  PROC DrawPart80()
    MoveL Offs(pOrigin,344.14,26.67,6.00),v60,z5,tPen\WObj:=wPaper;
    MoveL Offs(pOrigin,346.05,26.67,6.00),vTravel,z5,tPen\WObj:=wPaper;
    MoveL Offs(pOrigin,346.05,26.67,0.00),v60,z0,tPen\WObj:=wPaper;
    MoveL Offs(pOrigin,347.54,27.95,0.00),v40,z0,tPen\WObj:=wPaper;
    MoveL Offs(pOrigin,346.05,26.67,0.00),v40,fine,tPen\WObj:=wPaper;
    MoveL Offs(pOrigin,346.05,26.67,6.00),v60,z5,tPen\WObj:=wPaper;
    MoveL Offs(pOrigin,346.05,28.16,6.00),vTravel,z5,tPen\WObj:=wPaper;
    MoveL Offs(pOrigin,346.05,28.16,0.00),v60,z0,tPen\WObj:=wPaper;
    MoveL Offs(pOrigin,346.48,28.59,0.00),v40,z0,tPen\WObj:=wPaper;
    MoveL Offs(pOrigin,346.05,28.16,0.00),v40,fine,tPen\WObj:=wPaper;
    MoveL Offs(pOrigin,346.05,28.16,6.00),v60,z5,tPen\WObj:=wPaper;
    MoveL Offs(pOrigin,340.52,32.98,6.00),vTravel,z5,tPen\WObj:=wPaper;
    MoveL Offs(pOrigin,340.52,32.98,0.00),v60,z0,tPen\WObj:=wPaper;
    MoveL Offs(pOrigin,338.61,32.91,0.00),v40,z0,tPen\WObj:=wPaper;
    MoveL Offs(pOrigin,337.76,34.33,0.00),v40,z0,tPen\WObj:=wPaper;
    MoveL Offs(pOrigin,337.90,36.45,0.00),v40,z0,tPen\WObj:=wPaper;
    MoveL Offs(pOrigin,339.46,38.22,0.00),v40,z0,tPen\WObj:=wPaper;
    MoveL Offs(pOrigin,341.16,38.58,0.00),v40,z0,tPen\WObj:=wPaper;
    MoveL Offs(pOrigin,342.01,38.15,0.00),v40,z0,tPen\WObj:=wPaper;
    MoveL Offs(pOrigin,342.44,37.30,0.00),v40,z0,tPen\WObj:=wPaper;
    MoveL Offs(pOrigin,342.44,35.60,0.00),v40,z0,tPen\WObj:=wPaper;
    MoveL Offs(pOrigin,342.08,34.54,0.00),v40,z0,tPen\WObj:=wPaper;
    MoveL Offs(pOrigin,340.52,32.98,0.00),v40,fine,tPen\WObj:=wPaper;
    MoveL Offs(pOrigin,340.52,32.98,6.00),v60,z5,tPen\WObj:=wPaper;
    MoveL Offs(pOrigin,340.10,35.39,6.00),vTravel,z5,tPen\WObj:=wPaper;
    MoveL Offs(pOrigin,340.10,35.39,0.00),v60,z0,tPen\WObj:=wPaper;
    MoveL Offs(pOrigin,340.74,36.03,0.00),v40,fine,tPen\WObj:=wPaper;
    MoveL Offs(pOrigin,340.74,36.03,6.00),v60,z5,tPen\WObj:=wPaper;
    MoveL Offs(pOrigin,334.79,36.45,6.00),vTravel,z5,tPen\WObj:=wPaper;
    MoveL Offs(pOrigin,334.79,36.45,0.00),v60,z0,tPen\WObj:=wPaper;
    MoveL Offs(pOrigin,334.36,34.11,0.00),v40,z0,tPen\WObj:=wPaper;
    MoveL Offs(pOrigin,334.36,32.62,0.00),v40,z0,tPen\WObj:=wPaper;
    MoveL Offs(pOrigin,334.79,31.14,0.00),v40,fine,tPen\WObj:=wPaper;
    MoveL Offs(pOrigin,334.79,31.14,6.00),v60,z5,tPen\WObj:=wPaper;
    MoveL Offs(pOrigin,336.49,27.10,6.00),vTravel,z5,tPen\WObj:=wPaper;
    MoveL Offs(pOrigin,336.49,27.10,0.00),v60,z0,tPen\WObj:=wPaper;
    MoveL Offs(pOrigin,336.91,26.67,0.00),v40,z0,tPen\WObj:=wPaper;
    MoveL Offs(pOrigin,339.46,25.83,0.00),v40,z0,tPen\WObj:=wPaper;
    MoveL Offs(pOrigin,341.38,25.61,0.00),v40,z0,tPen\WObj:=wPaper;
    MoveL Offs(pOrigin,343.92,26.39,0.00),v40,z0,tPen\WObj:=wPaper;
    MoveL Offs(pOrigin,345.41,27.31,0.00),v40,z0,tPen\WObj:=wPaper;
    MoveL Offs(pOrigin,346.90,28.80,0.00),v40,z0,tPen\WObj:=wPaper;
    MoveL Offs(pOrigin,348.88,32.41,0.00),v40,z0,tPen\WObj:=wPaper;
    MoveL Offs(pOrigin,349.66,35.60,0.00),v40,z0,tPen\WObj:=wPaper;
    MoveL Offs(pOrigin,349.66,37.72,0.00),v40,z0,tPen\WObj:=wPaper;
    MoveL Offs(pOrigin,349.24,38.36,0.00),v40,z0,tPen\WObj:=wPaper;
    MoveL Offs(pOrigin,349.24,38.36,0.00),v40,z0,tPen\WObj:=wPaper;
    MoveL Offs(pOrigin,348.88,38.15,0.00),v40,z0,tPen\WObj:=wPaper;
    MoveL Offs(pOrigin,347.82,34.54,0.00),v40,z0,tPen\WObj:=wPaper;
    MoveL Offs(pOrigin,346.33,31.35,0.00),v40,z0,tPen\WObj:=wPaper;
    MoveL Offs(pOrigin,343.92,28.38,0.00),v40,z0,tPen\WObj:=wPaper;
    MoveL Offs(pOrigin,340.95,27.10,0.00),v40,z0,tPen\WObj:=wPaper;
    MoveL Offs(pOrigin,337.12,27.52,0.00),v40,z0,tPen\WObj:=wPaper;
    MoveL Offs(pOrigin,336.49,27.10,0.00),v40,fine,tPen\WObj:=wPaper;
    MoveL Offs(pOrigin,336.49,27.10,6.00),v60,z5,tPen\WObj:=wPaper;
    MoveL Offs(pOrigin,340.10,44.31,6.00),vTravel,z5,tPen\WObj:=wPaper;
    MoveL Offs(pOrigin,340.10,44.31,0.00),v60,z0,tPen\WObj:=wPaper;
    MoveL Offs(pOrigin,339.89,46.22,0.00),v40,z0,tPen\WObj:=wPaper;
    MoveL Offs(pOrigin,338.47,50.90,0.00),v40,z0,tPen\WObj:=wPaper;
    MoveL Offs(pOrigin,336.56,54.72,0.00),v40,z0,tPen\WObj:=wPaper;
    MoveL Offs(pOrigin,333.30,59.19,0.00),v40,z0,tPen\WObj:=wPaper;
    MoveL Offs(pOrigin,328.84,63.22,0.00),v40,fine,tPen\WObj:=wPaper;
    MoveL Offs(pOrigin,328.84,63.22,6.00),v60,z5,tPen\WObj:=wPaper;
    MoveL Offs(pOrigin,335.21,61.95,6.00),vTravel,z5,tPen\WObj:=wPaper;
    MoveL Offs(pOrigin,335.21,61.95,0.00),v60,z0,tPen\WObj:=wPaper;
    MoveL Offs(pOrigin,334.79,62.38,0.00),v40,z0,tPen\WObj:=wPaper;
    MoveL Offs(pOrigin,335.21,61.95,0.00),v40,fine,tPen\WObj:=wPaper;
    MoveL Offs(pOrigin,335.21,61.95,6.00),v60,z5,tPen\WObj:=wPaper;
    MoveL Offs(pOrigin,335.00,60.25,6.00),vTravel,z5,tPen\WObj:=wPaper;
    MoveL Offs(pOrigin,335.00,60.25,0.00),v60,z0,tPen\WObj:=wPaper;
    MoveL Offs(pOrigin,334.58,60.67,0.00),v40,z0,tPen\WObj:=wPaper;
    MoveL Offs(pOrigin,335.00,60.25,0.00),v40,fine,tPen\WObj:=wPaper;
    MoveL Offs(pOrigin,335.00,60.25,6.00),v60,z5,tPen\WObj:=wPaper;
    MoveL Offs(pOrigin,336.91,60.46,6.00),vTravel,z5,tPen\WObj:=wPaper;
    MoveL Offs(pOrigin,336.91,60.46,0.00),v60,z0,tPen\WObj:=wPaper;
    MoveL Offs(pOrigin,335.85,61.53,0.00),v40,z0,tPen\WObj:=wPaper;
    MoveL Offs(pOrigin,336.91,60.46,0.00),v40,fine,tPen\WObj:=wPaper;
    MoveL Offs(pOrigin,336.91,60.46,6.00),v60,z5,tPen\WObj:=wPaper;
    MoveL Offs(pOrigin,337.34,58.12,6.00),vTravel,z5,tPen\WObj:=wPaper;
    MoveL Offs(pOrigin,337.34,58.12,0.00),v60,z0,tPen\WObj:=wPaper;
    MoveL Offs(pOrigin,335.85,59.61,0.00),v40,z0,tPen\WObj:=wPaper;
    MoveL Offs(pOrigin,337.34,58.12,0.00),v40,fine,tPen\WObj:=wPaper;
    MoveL Offs(pOrigin,337.34,58.12,6.00),v60,z5,tPen\WObj:=wPaper;
    MoveL Offs(pOrigin,339.04,56.42,6.00),vTravel,z5,tPen\WObj:=wPaper;
    MoveL Offs(pOrigin,339.04,56.42,0.00),v60,z0,tPen\WObj:=wPaper;
    MoveL Offs(pOrigin,337.55,57.91,0.00),v40,z0,tPen\WObj:=wPaper;
    MoveL Offs(pOrigin,339.04,56.42,0.00),v40,z0,tPen\WObj:=wPaper;
    MoveL Offs(pOrigin,339.67,55.79,0.00),v40,z0,tPen\WObj:=wPaper;
    MoveL Offs(pOrigin,339.25,56.21,0.00),v40,z0,tPen\WObj:=wPaper;
    MoveL Offs(pOrigin,339.67,55.79,0.00),v40,fine,tPen\WObj:=wPaper;
    MoveL Offs(pOrigin,339.67,55.79,6.00),v60,z5,tPen\WObj:=wPaper;
    MoveL Offs(pOrigin,340.52,54.72,6.00),vTravel,z5,tPen\WObj:=wPaper;
    MoveL Offs(pOrigin,340.52,54.72,0.00),v60,z0,tPen\WObj:=wPaper;
    MoveL Offs(pOrigin,339.89,55.36,0.00),v40,z0,tPen\WObj:=wPaper;
    MoveL Offs(pOrigin,340.52,54.72,0.00),v40,fine,tPen\WObj:=wPaper;
    MoveL Offs(pOrigin,340.52,54.72,6.00),v60,z5,tPen\WObj:=wPaper;
    MoveL Offs(pOrigin,342.23,54.94,6.00),vTravel,z5,tPen\WObj:=wPaper;
    MoveL Offs(pOrigin,342.23,54.94,0.00),v60,z0,tPen\WObj:=wPaper;
    MoveL Offs(pOrigin,341.59,55.58,0.00),v40,z0,tPen\WObj:=wPaper;
    MoveL Offs(pOrigin,342.23,54.94,0.00),v40,fine,tPen\WObj:=wPaper;
    MoveL Offs(pOrigin,342.23,54.94,6.00),v60,z5,tPen\WObj:=wPaper;
    MoveL Offs(pOrigin,341.59,53.24,6.00),vTravel,z5,tPen\WObj:=wPaper;
    MoveL Offs(pOrigin,341.59,53.24,0.00),v60,z0,tPen\WObj:=wPaper;
    MoveL Offs(pOrigin,340.95,54.09,0.00),v40,z0,tPen\WObj:=wPaper;
    MoveL Offs(pOrigin,341.59,53.24,0.00),v40,fine,tPen\WObj:=wPaper;
    MoveL Offs(pOrigin,341.59,53.24,6.00),v60,z5,tPen\WObj:=wPaper;
    MoveL Offs(pOrigin,344.14,52.17,6.00),vTravel,z5,tPen\WObj:=wPaper;
    MoveL Offs(pOrigin,344.14,52.17,0.00),v60,z0,tPen\WObj:=wPaper;
    MoveL Offs(pOrigin,343.71,52.81,0.00),v40,z0,tPen\WObj:=wPaper;
    MoveL Offs(pOrigin,344.14,52.17,0.00),v40,fine,tPen\WObj:=wPaper;
    MoveL Offs(pOrigin,344.14,52.17,6.00),v60,z5,tPen\WObj:=wPaper;
    MoveL Offs(pOrigin,343.71,50.26,6.00),vTravel,z5,tPen\WObj:=wPaper;
    MoveL Offs(pOrigin,343.71,50.26,0.00),v60,z0,tPen\WObj:=wPaper;
    MoveL Offs(pOrigin,343.29,50.90,0.00),v40,z0,tPen\WObj:=wPaper;
    MoveL Offs(pOrigin,343.71,50.26,0.00),v40,fine,tPen\WObj:=wPaper;
    MoveL Offs(pOrigin,343.71,50.26,6.00),v60,z5,tPen\WObj:=wPaper;
    MoveL Offs(pOrigin,345.41,50.26,6.00),vTravel,z5,tPen\WObj:=wPaper;
    MoveL Offs(pOrigin,345.41,50.26,0.00),v60,z0,tPen\WObj:=wPaper;
    MoveL Offs(pOrigin,344.99,50.90,0.00),v40,z0,tPen\WObj:=wPaper;
    MoveL Offs(pOrigin,345.41,50.26,0.00),v40,fine,tPen\WObj:=wPaper;
  ENDPROC

  PROC DrawPart81()
    MoveL Offs(pOrigin,345.41,50.26,6.00),v60,z5,tPen\WObj:=wPaper;
    MoveL Offs(pOrigin,345.41,47.50,6.00),vTravel,z5,tPen\WObj:=wPaper;
    MoveL Offs(pOrigin,345.41,47.50,0.00),v60,z0,tPen\WObj:=wPaper;
    MoveL Offs(pOrigin,345.20,47.92,0.00),v40,z0,tPen\WObj:=wPaper;
    MoveL Offs(pOrigin,345.41,47.50,0.00),v40,fine,tPen\WObj:=wPaper;
    MoveL Offs(pOrigin,345.41,47.50,6.00),v60,z5,tPen\WObj:=wPaper;
    MoveL Offs(pOrigin,346.05,46.44,6.00),vTravel,z5,tPen\WObj:=wPaper;
    MoveL Offs(pOrigin,346.05,46.44,0.00),v60,z0,tPen\WObj:=wPaper;
    MoveL Offs(pOrigin,345.84,46.86,0.00),v40,z0,tPen\WObj:=wPaper;
    MoveL Offs(pOrigin,346.05,46.44,0.00),v40,fine,tPen\WObj:=wPaper;
    MoveL Offs(pOrigin,346.05,46.44,6.00),v60,z5,tPen\WObj:=wPaper;
    MoveL Offs(pOrigin,346.69,45.38,6.00),vTravel,z5,tPen\WObj:=wPaper;
    MoveL Offs(pOrigin,346.69,45.38,0.00),v60,z0,tPen\WObj:=wPaper;
    MoveL Offs(pOrigin,346.26,46.01,0.00),v40,z0,tPen\WObj:=wPaper;
    MoveL Offs(pOrigin,346.69,45.38,0.00),v40,z0,tPen\WObj:=wPaper;
    MoveL Offs(pOrigin,347.11,44.53,0.00),v40,z0,tPen\WObj:=wPaper;
    MoveL Offs(pOrigin,346.90,44.95,0.00),v40,z0,tPen\WObj:=wPaper;
    MoveL Offs(pOrigin,347.11,44.53,0.00),v40,fine,tPen\WObj:=wPaper;
    MoveL Offs(pOrigin,347.11,44.53,6.00),v60,z5,tPen\WObj:=wPaper;
    MoveL Offs(pOrigin,347.75,46.44,6.00),vTravel,z5,tPen\WObj:=wPaper;
    MoveL Offs(pOrigin,347.75,46.44,0.00),v60,z0,tPen\WObj:=wPaper;
    MoveL Offs(pOrigin,347.33,47.08,0.00),v40,z0,tPen\WObj:=wPaper;
    MoveL Offs(pOrigin,347.75,46.44,0.00),v40,fine,tPen\WObj:=wPaper;
    MoveL Offs(pOrigin,347.75,46.44,6.00),v60,z5,tPen\WObj:=wPaper;
    MoveL Offs(pOrigin,347.11,47.50,6.00),vTravel,z5,tPen\WObj:=wPaper;
    MoveL Offs(pOrigin,347.11,47.50,0.00),v60,z0,tPen\WObj:=wPaper;
    MoveL Offs(pOrigin,346.90,47.92,0.00),v40,z0,tPen\WObj:=wPaper;
    MoveL Offs(pOrigin,347.11,47.50,0.00),v40,fine,tPen\WObj:=wPaper;
    MoveL Offs(pOrigin,347.11,47.50,6.00),v60,z5,tPen\WObj:=wPaper;
    MoveL Offs(pOrigin,340.03,57.63,6.00),vTravel,z5,tPen\WObj:=wPaper;
    MoveL Offs(pOrigin,340.03,57.63,0.00),v60,z0,tPen\WObj:=wPaper;
    MoveL Offs(pOrigin,337.98,59.61,0.00),v40,z0,tPen\WObj:=wPaper;
    MoveL Offs(pOrigin,340.03,57.63,0.00),v40,fine,tPen\WObj:=wPaper;
    MoveL Offs(pOrigin,340.03,57.63,6.00),v60,z5,tPen\WObj:=wPaper;
    MoveL Offs(pOrigin,321.83,54.94,6.00),vTravel,z5,tPen\WObj:=wPaper;
    MoveL Offs(pOrigin,321.83,54.94,0.00),v60,z0,tPen\WObj:=wPaper;
    MoveL Offs(pOrigin,321.61,55.36,0.00),v40,z0,tPen\WObj:=wPaper;
    MoveL Offs(pOrigin,321.83,54.94,0.00),v40,fine,tPen\WObj:=wPaper;
    MoveL Offs(pOrigin,321.83,54.94,6.00),v60,z5,tPen\WObj:=wPaper;
    MoveL Offs(pOrigin,321.19,56.21,6.00),vTravel,z5,tPen\WObj:=wPaper;
    MoveL Offs(pOrigin,321.19,56.21,0.00),v60,z0,tPen\WObj:=wPaper;
    MoveL Offs(pOrigin,320.98,56.64,0.00),v40,z0,tPen\WObj:=wPaper;
    MoveL Offs(pOrigin,321.19,56.21,0.00),v40,fine,tPen\WObj:=wPaper;
    MoveL Offs(pOrigin,321.19,56.21,6.00),v60,z5,tPen\WObj:=wPaper;
    MoveL Offs(pOrigin,319.70,58.76,6.00),vTravel,z5,tPen\WObj:=wPaper;
    MoveL Offs(pOrigin,319.70,58.76,0.00),v60,z0,tPen\WObj:=wPaper;
    MoveL Offs(pOrigin,319.91,58.34,0.00),v40,z0,tPen\WObj:=wPaper;
    MoveL Offs(pOrigin,319.70,58.76,0.00),v40,fine,tPen\WObj:=wPaper;
    MoveL Offs(pOrigin,319.70,58.76,6.00),v60,z5,tPen\WObj:=wPaper;
    MoveL Offs(pOrigin,318.85,59.61,6.00),vTravel,z5,tPen\WObj:=wPaper;
    MoveL Offs(pOrigin,318.85,59.61,0.00),v60,z0,tPen\WObj:=wPaper;
    MoveL Offs(pOrigin,318.64,60.04,0.00),v40,z0,tPen\WObj:=wPaper;
    MoveL Offs(pOrigin,318.85,59.61,0.00),v40,fine,tPen\WObj:=wPaper;
    MoveL Offs(pOrigin,318.85,59.61,6.00),v60,z5,tPen\WObj:=wPaper;
    MoveL Offs(pOrigin,317.58,57.28,6.00),vTravel,z5,tPen\WObj:=wPaper;
    MoveL Offs(pOrigin,317.58,57.28,0.00),v60,z0,tPen\WObj:=wPaper;
    MoveL Offs(pOrigin,316.94,57.91,0.00),v40,z0,tPen\WObj:=wPaper;
    MoveL Offs(pOrigin,317.58,57.28,0.00),v40,fine,tPen\WObj:=wPaper;
    MoveL Offs(pOrigin,317.58,57.28,6.00),v60,z5,tPen\WObj:=wPaper;
    MoveL Offs(pOrigin,316.09,58.76,6.00),vTravel,z5,tPen\WObj:=wPaper;
    MoveL Offs(pOrigin,316.09,58.76,0.00),v60,z0,tPen\WObj:=wPaper;
    MoveL Offs(pOrigin,315.66,59.19,0.00),v40,z0,tPen\WObj:=wPaper;
    MoveL Offs(pOrigin,316.09,58.76,0.00),v40,fine,tPen\WObj:=wPaper;
    MoveL Offs(pOrigin,316.09,58.76,6.00),v60,z5,tPen\WObj:=wPaper;
    MoveL Offs(pOrigin,313.11,61.74,6.00),vTravel,z5,tPen\WObj:=wPaper;
    MoveL Offs(pOrigin,313.11,61.74,0.00),v60,z0,tPen\WObj:=wPaper;
    MoveL Offs(pOrigin,311.41,61.53,0.00),v40,fine,tPen\WObj:=wPaper;
    MoveL Offs(pOrigin,311.41,61.53,6.00),v60,z5,tPen\WObj:=wPaper;
    MoveL Offs(pOrigin,309.29,62.38,6.00),vTravel,z5,tPen\WObj:=wPaper;
    MoveL Offs(pOrigin,309.29,62.38,0.00),v60,z0,tPen\WObj:=wPaper;
    MoveL Offs(pOrigin,308.86,61.88,0.00),v40,z0,tPen\WObj:=wPaper;
    MoveL Offs(pOrigin,305.89,60.89,0.00),v40,z0,tPen\WObj:=wPaper;
    MoveL Offs(pOrigin,303.34,61.53,0.00),v40,z0,tPen\WObj:=wPaper;
    MoveL Offs(pOrigin,303.34,61.53,0.00),v40,z0,tPen\WObj:=wPaper;
    MoveL Offs(pOrigin,303.76,62.09,0.00),v40,z0,tPen\WObj:=wPaper;
    MoveL Offs(pOrigin,305.67,62.59,0.00),v40,z0,tPen\WObj:=wPaper;
    MoveL Offs(pOrigin,308.65,62.80,0.00),v40,z0,tPen\WObj:=wPaper;
    MoveL Offs(pOrigin,309.29,62.38,0.00),v40,fine,tPen\WObj:=wPaper;
    MoveL Offs(pOrigin,309.29,62.38,6.00),v60,z5,tPen\WObj:=wPaper;
    MoveL Offs(pOrigin,312.48,69.18,6.00),vTravel,z5,tPen\WObj:=wPaper;
    MoveL Offs(pOrigin,312.48,69.18,0.00),v60,z0,tPen\WObj:=wPaper;
    MoveL Offs(pOrigin,312.90,69.39,0.00),v40,z0,tPen\WObj:=wPaper;
    MoveL Offs(pOrigin,312.48,69.18,0.00),v40,z0,tPen\WObj:=wPaper;
    MoveL Offs(pOrigin,313.33,69.60,0.00),v40,z0,tPen\WObj:=wPaper;
    MoveL Offs(pOrigin,313.75,69.81,0.00),v40,z0,tPen\WObj:=wPaper;
    MoveL Offs(pOrigin,313.33,69.60,0.00),v40,fine,tPen\WObj:=wPaper;
    MoveL Offs(pOrigin,313.33,69.60,6.00),v60,z5,tPen\WObj:=wPaper;
    MoveL Offs(pOrigin,314.17,68.11,6.00),vTravel,z5,tPen\WObj:=wPaper;
    MoveL Offs(pOrigin,314.17,68.11,0.00),v60,z0,tPen\WObj:=wPaper;
    MoveL Offs(pOrigin,316.30,68.75,0.00),v40,fine,tPen\WObj:=wPaper;
    MoveL Offs(pOrigin,316.30,68.75,6.00),v60,z5,tPen\WObj:=wPaper;
    MoveL Offs(pOrigin,320.34,52.39,6.00),vTravel,z5,tPen\WObj:=wPaper;
    MoveL Offs(pOrigin,320.34,52.39,0.00),v60,z0,tPen\WObj:=wPaper;
    MoveL Offs(pOrigin,320.90,50.26,0.00),v40,z0,tPen\WObj:=wPaper;
    MoveL Offs(pOrigin,321.61,49.20,0.00),v40,z0,tPen\WObj:=wPaper;
    MoveL Offs(pOrigin,321.61,49.20,0.00),v40,z0,tPen\WObj:=wPaper;
    MoveL Offs(pOrigin,321.61,48.14,0.00),v40,z0,tPen\WObj:=wPaper;
    MoveL Offs(pOrigin,322.25,47.92,0.00),v40,fine,tPen\WObj:=wPaper;
    MoveL Offs(pOrigin,322.25,47.92,6.00),v60,z5,tPen\WObj:=wPaper;
    MoveL Offs(pOrigin,308.65,48.99,6.00),vTravel,z5,tPen\WObj:=wPaper;
    MoveL Offs(pOrigin,308.65,48.99,0.00),v60,z0,tPen\WObj:=wPaper;
    MoveL Offs(pOrigin,307.02,52.60,0.00),v40,z0,tPen\WObj:=wPaper;
    MoveL Offs(pOrigin,304.19,56.42,0.00),v40,fine,tPen\WObj:=wPaper;
    MoveL Offs(pOrigin,304.19,56.42,6.00),v60,z5,tPen\WObj:=wPaper;
    MoveL Offs(pOrigin,291.23,65.35,6.00),vTravel,z5,tPen\WObj:=wPaper;
    MoveL Offs(pOrigin,291.23,65.35,0.00),v60,z0,tPen\WObj:=wPaper;
    MoveL Offs(pOrigin,291.65,65.14,0.00),v40,z0,tPen\WObj:=wPaper;
    MoveL Offs(pOrigin,291.23,65.35,0.00),v40,fine,tPen\WObj:=wPaper;
    MoveL Offs(pOrigin,291.23,65.35,6.00),v60,z5,tPen\WObj:=wPaper;
    MoveL Offs(pOrigin,271.67,79.59,6.00),vTravel,z5,tPen\WObj:=wPaper;
    MoveL Offs(pOrigin,271.67,79.59,0.00),v60,z0,tPen\WObj:=wPaper;
    MoveL Offs(pOrigin,267.42,73.64,0.00),v40,z0,tPen\WObj:=wPaper;
    MoveL Offs(pOrigin,259.14,64.93,0.00),v40,fine,tPen\WObj:=wPaper;
    MoveL Offs(pOrigin,259.14,64.93,6.00),v60,z5,tPen\WObj:=wPaper;
    MoveL Offs(pOrigin,261.48,71.30,6.00),vTravel,z5,tPen\WObj:=wPaper;
    MoveL Offs(pOrigin,261.48,71.30,0.00),v60,z0,tPen\WObj:=wPaper;
    MoveL Offs(pOrigin,265.73,76.40,0.00),v40,z0,tPen\WObj:=wPaper;
    MoveL Offs(pOrigin,269.55,82.14,0.00),v40,fine,tPen\WObj:=wPaper;
    MoveL Offs(pOrigin,269.55,82.14,6.00),v60,z5,tPen\WObj:=wPaper;
    MoveL Offs(pOrigin,270.83,78.53,6.00),vTravel,z5,tPen\WObj:=wPaper;
  ENDPROC

  PROC DrawPart82()
    MoveL Offs(pOrigin,270.83,78.53,0.00),v60,z0,tPen\WObj:=wPaper;
    MoveL Offs(pOrigin,271.04,78.95,0.00),v40,z0,tPen\WObj:=wPaper;
    MoveL Offs(pOrigin,270.83,78.53,0.00),v40,fine,tPen\WObj:=wPaper;
    MoveL Offs(pOrigin,270.83,78.53,6.00),v60,z5,tPen\WObj:=wPaper;
    MoveL Offs(pOrigin,269.76,76.82,6.00),vTravel,z5,tPen\WObj:=wPaper;
    MoveL Offs(pOrigin,269.76,76.82,0.00),v60,z0,tPen\WObj:=wPaper;
    MoveL Offs(pOrigin,270.19,77.46,0.00),v40,z0,tPen\WObj:=wPaper;
    MoveL Offs(pOrigin,269.76,76.82,0.00),v40,z0,tPen\WObj:=wPaper;
    MoveL Offs(pOrigin,269.12,75.97,0.00),v40,z0,tPen\WObj:=wPaper;
    MoveL Offs(pOrigin,269.55,76.61,0.00),v40,z0,tPen\WObj:=wPaper;
    MoveL Offs(pOrigin,269.12,75.97,0.00),v40,fine,tPen\WObj:=wPaper;
    MoveL Offs(pOrigin,269.12,75.97,6.00),v60,z5,tPen\WObj:=wPaper;
    MoveL Offs(pOrigin,267.85,74.49,6.00),vTravel,z5,tPen\WObj:=wPaper;
    MoveL Offs(pOrigin,267.85,74.49,0.00),v60,z0,tPen\WObj:=wPaper;
    MoveL Offs(pOrigin,268.49,75.12,0.00),v40,z0,tPen\WObj:=wPaper;
    MoveL Offs(pOrigin,267.85,74.49,0.00),v40,fine,tPen\WObj:=wPaper;
    MoveL Offs(pOrigin,267.85,74.49,6.00),v60,z5,tPen\WObj:=wPaper;
    MoveL Offs(pOrigin,266.58,73.00,6.00),vTravel,z5,tPen\WObj:=wPaper;
    MoveL Offs(pOrigin,266.58,73.00,0.00),v60,z0,tPen\WObj:=wPaper;
    MoveL Offs(pOrigin,267.42,73.85,0.00),v40,z0,tPen\WObj:=wPaper;
    MoveL Offs(pOrigin,266.58,73.00,0.00),v40,fine,tPen\WObj:=wPaper;
    MoveL Offs(pOrigin,266.58,73.00,6.00),v60,z5,tPen\WObj:=wPaper;
    MoveL Offs(pOrigin,265.30,71.51,6.00),vTravel,z5,tPen\WObj:=wPaper;
    MoveL Offs(pOrigin,265.30,71.51,0.00),v60,z0,tPen\WObj:=wPaper;
    MoveL Offs(pOrigin,265.94,72.15,0.00),v40,z0,tPen\WObj:=wPaper;
    MoveL Offs(pOrigin,265.30,71.51,0.00),v40,fine,tPen\WObj:=wPaper;
    MoveL Offs(pOrigin,265.30,71.51,6.00),v60,z5,tPen\WObj:=wPaper;
    MoveL Offs(pOrigin,258.50,33.90,6.00),vTravel,z5,tPen\WObj:=wPaper;
    MoveL Offs(pOrigin,258.50,33.90,0.00),v60,z0,tPen\WObj:=wPaper;
    MoveL Offs(pOrigin,257.65,33.83,0.00),v40,z0,tPen\WObj:=wPaper;
    MoveL Offs(pOrigin,256.16,32.84,0.00),v40,z0,tPen\WObj:=wPaper;
    MoveL Offs(pOrigin,255.38,31.99,0.00),v40,z0,tPen\WObj:=wPaper;
    MoveL Offs(pOrigin,255.31,31.35,0.00),v40,z0,tPen\WObj:=wPaper;
    MoveL Offs(pOrigin,255.74,30.50,0.00),v40,z0,tPen\WObj:=wPaper;
    MoveL Offs(pOrigin,257.23,29.30,0.00),v40,z0,tPen\WObj:=wPaper;
    MoveL Offs(pOrigin,259.77,29.44,0.00),v40,fine,tPen\WObj:=wPaper;
    MoveL Offs(pOrigin,259.77,29.44,6.00),v60,z5,tPen\WObj:=wPaper;
    MoveL Offs(pOrigin,255.95,30.08,6.00),vTravel,z5,tPen\WObj:=wPaper;
    MoveL Offs(pOrigin,255.95,30.08,0.00),v60,z0,tPen\WObj:=wPaper;
    MoveL Offs(pOrigin,255.52,30.50,0.00),v40,z0,tPen\WObj:=wPaper;
    MoveL Offs(pOrigin,255.95,30.08,0.00),v40,fine,tPen\WObj:=wPaper;
    MoveL Offs(pOrigin,255.95,30.08,6.00),v60,z5,tPen\WObj:=wPaper;
    MoveL Offs(pOrigin,255.31,32.20,6.00),vTravel,z5,tPen\WObj:=wPaper;
    MoveL Offs(pOrigin,255.31,32.20,0.00),v60,z0,tPen\WObj:=wPaper;
    MoveL Offs(pOrigin,256.16,33.05,0.00),v40,z0,tPen\WObj:=wPaper;
    MoveL Offs(pOrigin,255.31,32.20,0.00),v40,fine,tPen\WObj:=wPaper;
    MoveL Offs(pOrigin,255.31,32.20,6.00),v60,z5,tPen\WObj:=wPaper;
    MoveL Offs(pOrigin,257.65,21.58,6.00),vTravel,z5,tPen\WObj:=wPaper;
    MoveL Offs(pOrigin,257.65,21.58,0.00),v60,z0,tPen\WObj:=wPaper;
    MoveL Offs(pOrigin,259.35,22.00,0.00),v40,z0,tPen\WObj:=wPaper;
    MoveL Offs(pOrigin,259.35,22.00,0.00),v40,z0,tPen\WObj:=wPaper;
    MoveL Offs(pOrigin,259.56,21.36,0.00),v40,z0,tPen\WObj:=wPaper;
    MoveL Offs(pOrigin,260.20,21.58,0.00),v40,z0,tPen\WObj:=wPaper;
    MoveL Offs(pOrigin,260.20,21.58,0.00),v40,z0,tPen\WObj:=wPaper;
    MoveL Offs(pOrigin,264.24,22.64,0.00),v40,z0,tPen\WObj:=wPaper;
    MoveL Offs(pOrigin,264.24,23.27,0.00),v40,z0,tPen\WObj:=wPaper;
    MoveL Offs(pOrigin,260.20,22.21,0.00),v40,fine,tPen\WObj:=wPaper;
    MoveL Offs(pOrigin,260.20,22.21,6.00),v60,z5,tPen\WObj:=wPaper;
    MoveL Offs(pOrigin,259.35,21.36,6.00),vTravel,z5,tPen\WObj:=wPaper;
    MoveL Offs(pOrigin,259.35,21.36,0.00),v60,z0,tPen\WObj:=wPaper;
    MoveL Offs(pOrigin,257.65,20.94,0.00),v40,z0,tPen\WObj:=wPaper;
    MoveL Offs(pOrigin,256.80,20.73,0.00),v40,z0,tPen\WObj:=wPaper;
    MoveL Offs(pOrigin,251.27,19.24,0.00),v40,z0,tPen\WObj:=wPaper;
    MoveL Offs(pOrigin,251.27,19.88,0.00),v40,z0,tPen\WObj:=wPaper;
    MoveL Offs(pOrigin,256.80,21.36,0.00),v40,fine,tPen\WObj:=wPaper;
    MoveL Offs(pOrigin,256.80,21.36,6.00),v60,z5,tPen\WObj:=wPaper;
    MoveL Offs(pOrigin,250.43,19.66,6.00),vTravel,z5,tPen\WObj:=wPaper;
    MoveL Offs(pOrigin,250.43,19.66,0.00),v60,z0,tPen\WObj:=wPaper;
    MoveL Offs(pOrigin,233.64,15.41,0.00),v40,z0,tPen\WObj:=wPaper;
    MoveL Offs(pOrigin,210.26,17.54,0.00),v40,z0,tPen\WObj:=wPaper;
    MoveL Offs(pOrigin,209.70,17.96,0.00),v40,z0,tPen\WObj:=wPaper;
    MoveL Offs(pOrigin,210.26,19.38,0.00),v40,z0,tPen\WObj:=wPaper;
    MoveL Offs(pOrigin,212.39,19.45,0.00),v40,z0,tPen\WObj:=wPaper;
    MoveL Offs(pOrigin,234.06,17.33,0.00),v40,z0,tPen\WObj:=wPaper;
    MoveL Offs(pOrigin,273.16,27.10,0.00),v40,z0,tPen\WObj:=wPaper;
    MoveL Offs(pOrigin,273.80,26.89,0.00),v40,z0,tPen\WObj:=wPaper;
    MoveL Offs(pOrigin,274.01,26.04,0.00),v40,z0,tPen\WObj:=wPaper;
    MoveL Offs(pOrigin,273.38,25.61,0.00),v40,z0,tPen\WObj:=wPaper;
    MoveL Offs(pOrigin,273.38,24.98,0.00),v40,z0,tPen\WObj:=wPaper;
    MoveL Offs(pOrigin,274.86,25.12,0.00),v40,z0,tPen\WObj:=wPaper;
    MoveL Offs(pOrigin,275.29,23.91,0.00),v40,z0,tPen\WObj:=wPaper;
    MoveL Offs(pOrigin,274.01,23.27,0.00),v40,z0,tPen\WObj:=wPaper;
    MoveL Offs(pOrigin,234.91,13.07,0.00),v40,z0,tPen\WObj:=wPaper;
    MoveL Offs(pOrigin,230.45,13.07,0.00),v40,z0,tPen\WObj:=wPaper;
    MoveL Offs(pOrigin,210.26,15.20,0.00),v40,z0,tPen\WObj:=wPaper;
    MoveL Offs(pOrigin,209.62,15.84,0.00),v40,z0,tPen\WObj:=wPaper;
    MoveL Offs(pOrigin,210.05,16.48,0.00),v40,z0,tPen\WObj:=wPaper;
    MoveL Offs(pOrigin,212.39,16.48,0.00),v40,z0,tPen\WObj:=wPaper;
    MoveL Offs(pOrigin,230.45,14.56,0.00),v40,z0,tPen\WObj:=wPaper;
    MoveL Offs(pOrigin,233.64,14.56,0.00),v40,z0,tPen\WObj:=wPaper;
    MoveL Offs(pOrigin,250.43,19.02,0.00),v40,fine,tPen\WObj:=wPaper;
    MoveL Offs(pOrigin,250.43,19.02,6.00),v60,z5,tPen\WObj:=wPaper;
    MoveL Offs(pOrigin,265.09,22.85,6.00),vTravel,z5,tPen\WObj:=wPaper;
    MoveL Offs(pOrigin,265.09,22.85,0.00),v60,z0,tPen\WObj:=wPaper;
    MoveL Offs(pOrigin,268.27,23.70,0.00),v40,z0,tPen\WObj:=wPaper;
    MoveL Offs(pOrigin,268.27,24.34,0.00),v40,z0,tPen\WObj:=wPaper;
    MoveL Offs(pOrigin,265.09,23.49,0.00),v40,fine,tPen\WObj:=wPaper;
    MoveL Offs(pOrigin,265.09,23.49,6.00),v60,z5,tPen\WObj:=wPaper;
    MoveL Offs(pOrigin,269.12,24.55,6.00),vTravel,z5,tPen\WObj:=wPaper;
    MoveL Offs(pOrigin,269.12,24.55,0.00),v60,z0,tPen\WObj:=wPaper;
    MoveL Offs(pOrigin,270.83,24.98,0.00),v40,z0,tPen\WObj:=wPaper;
    MoveL Offs(pOrigin,270.83,24.34,0.00),v40,z0,tPen\WObj:=wPaper;
    MoveL Offs(pOrigin,269.34,23.91,0.00),v40,z0,tPen\WObj:=wPaper;
    MoveL Offs(pOrigin,269.12,24.55,0.00),v40,fine,tPen\WObj:=wPaper;
    MoveL Offs(pOrigin,269.12,24.55,6.00),v60,z5,tPen\WObj:=wPaper;
    MoveL Offs(pOrigin,272.52,25.40,6.00),vTravel,z5,tPen\WObj:=wPaper;
    MoveL Offs(pOrigin,272.52,25.40,0.00),v60,z0,tPen\WObj:=wPaper;
    MoveL Offs(pOrigin,272.74,24.76,0.00),v40,z0,tPen\WObj:=wPaper;
    MoveL Offs(pOrigin,273.38,24.98,0.00),v40,fine,tPen\WObj:=wPaper;
    MoveL Offs(pOrigin,273.38,24.98,6.00),v60,z5,tPen\WObj:=wPaper;
    MoveL Offs(pOrigin,275.08,24.55,6.00),vTravel,z5,tPen\WObj:=wPaper;
    MoveL Offs(pOrigin,275.08,24.55,0.00),v60,z0,tPen\WObj:=wPaper;
    MoveL Offs(pOrigin,274.86,24.98,0.00),v40,z0,tPen\WObj:=wPaper;
    MoveL Offs(pOrigin,275.08,24.55,0.00),v40,fine,tPen\WObj:=wPaper;
    MoveL Offs(pOrigin,275.08,24.55,6.00),v60,z5,tPen\WObj:=wPaper;
    MoveL Offs(pOrigin,275.50,26.46,6.00),vTravel,z5,tPen\WObj:=wPaper;
    MoveL Offs(pOrigin,275.50,26.46,0.00),v60,z0,tPen\WObj:=wPaper;
    MoveL Offs(pOrigin,275.29,26.89,0.00),v40,z0,tPen\WObj:=wPaper;
    MoveL Offs(pOrigin,275.50,26.46,0.00),v40,fine,tPen\WObj:=wPaper;
    MoveL Offs(pOrigin,275.50,26.46,6.00),v60,z5,tPen\WObj:=wPaper;
  ENDPROC

  PROC DrawPart83()
    MoveL Offs(pOrigin,295.48,26.67,6.00),vTravel,z5,tPen\WObj:=wPaper;
    MoveL Offs(pOrigin,295.48,26.67,0.00),v60,z0,tPen\WObj:=wPaper;
    MoveL Offs(pOrigin,295.69,27.10,0.00),v40,z0,tPen\WObj:=wPaper;
    MoveL Offs(pOrigin,295.48,26.67,0.00),v40,fine,tPen\WObj:=wPaper;
    MoveL Offs(pOrigin,295.48,26.67,6.00),v60,z5,tPen\WObj:=wPaper;
    MoveL Offs(pOrigin,338.19,83.41,6.00),vTravel,z5,tPen\WObj:=wPaper;
    MoveL Offs(pOrigin,338.19,83.41,0.00),v60,z0,tPen\WObj:=wPaper;
    MoveL Offs(pOrigin,338.40,83.84,0.00),v40,z0,tPen\WObj:=wPaper;
    MoveL Offs(pOrigin,338.19,83.41,0.00),v40,fine,tPen\WObj:=wPaper;
    MoveL Offs(pOrigin,338.19,83.41,6.00),v60,z5,tPen\WObj:=wPaper;
    MoveL Offs(pOrigin,350.30,90.64,6.00),vTravel,z5,tPen\WObj:=wPaper;
    MoveL Offs(pOrigin,350.30,90.64,0.00),v60,z0,tPen\WObj:=wPaper;
    MoveL Offs(pOrigin,348.60,77.25,0.00),v40,z0,tPen\WObj:=wPaper;
    MoveL Offs(pOrigin,348.81,76.82,0.00),v40,z0,tPen\WObj:=wPaper;
    MoveL Offs(pOrigin,351.36,77.04,0.00),v40,z0,tPen\WObj:=wPaper;
    MoveL Offs(pOrigin,352.42,77.46,0.00),v40,z0,tPen\WObj:=wPaper;
    MoveL Offs(pOrigin,351.79,82.35,0.00),v40,z0,tPen\WObj:=wPaper;
    MoveL Offs(pOrigin,351.58,87.66,0.00),v40,z0,tPen\WObj:=wPaper;
    MoveL Offs(pOrigin,350.94,90.21,0.00),v40,z0,tPen\WObj:=wPaper;
    MoveL Offs(pOrigin,350.30,91.28,0.00),v40,fine,tPen\WObj:=wPaper;
    MoveL Offs(pOrigin,350.30,91.28,6.00),v60,z5,tPen\WObj:=wPaper;
    MoveL Offs(pOrigin,351.36,92.97,6.00),vTravel,z5,tPen\WObj:=wPaper;
    MoveL Offs(pOrigin,351.36,92.97,0.00),v60,z0,tPen\WObj:=wPaper;
    MoveL Offs(pOrigin,350.94,93.61,0.00),v40,z0,tPen\WObj:=wPaper;
    MoveL Offs(pOrigin,351.36,92.97,0.00),v40,z0,tPen\WObj:=wPaper;
    MoveL Offs(pOrigin,350.73,93.82,0.00),v40,z0,tPen\WObj:=wPaper;
    MoveL Offs(pOrigin,350.30,94.46,0.00),v40,z0,tPen\WObj:=wPaper;
    MoveL Offs(pOrigin,350.73,93.82,0.00),v40,fine,tPen\WObj:=wPaper;
    MoveL Offs(pOrigin,350.73,93.82,6.00),v60,z5,tPen\WObj:=wPaper;
    MoveL Offs(pOrigin,348.39,94.46,6.00),vTravel,z5,tPen\WObj:=wPaper;
    MoveL Offs(pOrigin,348.39,94.46,0.00),v60,z0,tPen\WObj:=wPaper;
    MoveL Offs(pOrigin,347.96,95.10,0.00),v40,z0,tPen\WObj:=wPaper;
    MoveL Offs(pOrigin,348.39,94.46,0.00),v40,fine,tPen\WObj:=wPaper;
    MoveL Offs(pOrigin,348.39,94.46,6.00),v60,z5,tPen\WObj:=wPaper;
    MoveL Offs(pOrigin,352.42,91.91,6.00),vTravel,z5,tPen\WObj:=wPaper;
    MoveL Offs(pOrigin,352.42,91.91,0.00),v60,z0,tPen\WObj:=wPaper;
    MoveL Offs(pOrigin,352.42,91.28,0.00),v40,z0,tPen\WObj:=wPaper;
    MoveL Offs(pOrigin,353.27,91.28,0.00),v40,z0,tPen\WObj:=wPaper;
    MoveL Offs(pOrigin,353.27,91.28,0.00),v40,z0,tPen\WObj:=wPaper;
    MoveL Offs(pOrigin,353.49,92.12,0.00),v40,z0,tPen\WObj:=wPaper;
    MoveL Offs(pOrigin,353.06,92.34,0.00),v40,z0,tPen\WObj:=wPaper;
    MoveL Offs(pOrigin,353.06,92.34,0.00),v40,z0,tPen\WObj:=wPaper;
    MoveL Offs(pOrigin,354.05,95.74,0.00),v40,z0,tPen\WObj:=wPaper;
    MoveL Offs(pOrigin,355.12,97.86,0.00),v40,z0,tPen\WObj:=wPaper;
    MoveL Offs(pOrigin,357.74,101.47,0.00),v40,fine,tPen\WObj:=wPaper;
    MoveL Offs(pOrigin,357.74,101.47,6.00),v60,z5,tPen\WObj:=wPaper;
    MoveL Offs(pOrigin,356.04,104.03,6.00),vTravel,z5,tPen\WObj:=wPaper;
    MoveL Offs(pOrigin,356.04,104.03,0.00),v60,z0,tPen\WObj:=wPaper;
    MoveL Offs(pOrigin,364.11,107.21,0.00),v40,z0,tPen\WObj:=wPaper;
    MoveL Offs(pOrigin,370.70,108.49,0.00),v40,z0,tPen\WObj:=wPaper;
    MoveL Offs(pOrigin,370.70,108.49,0.00),v40,z0,tPen\WObj:=wPaper;
    MoveL Offs(pOrigin,371.12,108.91,0.00),v40,z0,tPen\WObj:=wPaper;
    MoveL Offs(pOrigin,371.98,108.70,0.00),v40,z0,tPen\WObj:=wPaper;
    MoveL Offs(pOrigin,371.98,108.70,0.00),v40,z0,tPen\WObj:=wPaper;
    MoveL Offs(pOrigin,371.55,108.06,0.00),v40,z0,tPen\WObj:=wPaper;
    MoveL Offs(pOrigin,370.91,108.06,0.00),v40,z0,tPen\WObj:=wPaper;
    MoveL Offs(pOrigin,370.70,108.49,0.00),v40,fine,tPen\WObj:=wPaper;
    MoveL Offs(pOrigin,370.70,108.49,6.00),v60,z5,tPen\WObj:=wPaper;
    MoveL Offs(pOrigin,371.98,108.70,6.00),vTravel,z5,tPen\WObj:=wPaper;
    MoveL Offs(pOrigin,371.98,108.70,0.00),v60,z0,tPen\WObj:=wPaper;
    MoveL Offs(pOrigin,377.92,108.70,0.00),v40,z0,tPen\WObj:=wPaper;
    MoveL Offs(pOrigin,382.60,108.06,0.00),v40,z0,tPen\WObj:=wPaper;
    MoveL Offs(pOrigin,389.61,106.36,0.00),v40,z0,tPen\WObj:=wPaper;
    MoveL Offs(pOrigin,394.50,104.45,0.00),v40,fine,tPen\WObj:=wPaper;
    MoveL Offs(pOrigin,394.50,104.45,6.00),v60,z5,tPen\WObj:=wPaper;
    MoveL Offs(pOrigin,393.44,100.84,6.00),vTravel,z5,tPen\WObj:=wPaper;
    MoveL Offs(pOrigin,393.44,100.84,0.00),v60,z0,tPen\WObj:=wPaper;
    MoveL Offs(pOrigin,384.51,103.39,0.00),v40,z0,tPen\WObj:=wPaper;
    MoveL Offs(pOrigin,379.20,104.24,0.00),v40,z0,tPen\WObj:=wPaper;
    MoveL Offs(pOrigin,371.55,104.24,0.00),v40,z0,tPen\WObj:=wPaper;
    MoveL Offs(pOrigin,365.39,102.75,0.00),v40,z0,tPen\WObj:=wPaper;
    MoveL Offs(pOrigin,365.39,102.75,0.00),v40,z0,tPen\WObj:=wPaper;
    MoveL Offs(pOrigin,365.60,103.39,0.00),v40,z0,tPen\WObj:=wPaper;
    MoveL Offs(pOrigin,366.66,103.88,0.00),v40,z0,tPen\WObj:=wPaper;
    MoveL Offs(pOrigin,371.55,105.09,0.00),v40,z0,tPen\WObj:=wPaper;
    MoveL Offs(pOrigin,377.71,105.30,0.00),v40,z0,tPen\WObj:=wPaper;
    MoveL Offs(pOrigin,381.54,104.88,0.00),v40,z0,tPen\WObj:=wPaper;
    MoveL Offs(pOrigin,388.12,103.39,0.00),v40,z0,tPen\WObj:=wPaper;
    MoveL Offs(pOrigin,392.80,101.76,0.00),v40,z0,tPen\WObj:=wPaper;
    MoveL Offs(pOrigin,393.86,100.77,0.00),v40,z0,tPen\WObj:=wPaper;
    MoveL Offs(pOrigin,396.84,99.42,0.00),v40,z0,tPen\WObj:=wPaper;
    MoveL Offs(pOrigin,400.10,97.30,0.00),v40,z0,tPen\WObj:=wPaper;
    MoveL Offs(pOrigin,399.81,97.44,0.00),v40,z0,tPen\WObj:=wPaper;
    MoveL Offs(pOrigin,400.66,97.01,0.00),v40,z0,tPen\WObj:=wPaper;
    MoveL Offs(pOrigin,404.49,93.61,0.00),v40,fine,tPen\WObj:=wPaper;
    MoveL Offs(pOrigin,404.49,93.61,6.00),v60,z5,tPen\WObj:=wPaper;
    MoveL Offs(pOrigin,404.91,98.93,6.00),vTravel,z5,tPen\WObj:=wPaper;
    MoveL Offs(pOrigin,404.91,98.93,0.00),v60,z0,tPen\WObj:=wPaper;
    MoveL Offs(pOrigin,404.70,99.35,0.00),v40,z0,tPen\WObj:=wPaper;
    MoveL Offs(pOrigin,404.91,98.93,0.00),v40,z0,tPen\WObj:=wPaper;
    MoveL Offs(pOrigin,404.49,99.78,0.00),v40,z0,tPen\WObj:=wPaper;
    MoveL Offs(pOrigin,404.27,100.20,0.00),v40,z0,tPen\WObj:=wPaper;
    MoveL Offs(pOrigin,404.49,99.78,0.00),v40,fine,tPen\WObj:=wPaper;
    MoveL Offs(pOrigin,404.49,99.78,6.00),v60,z5,tPen\WObj:=wPaper;
    MoveL Offs(pOrigin,403.85,100.84,6.00),vTravel,z5,tPen\WObj:=wPaper;
    MoveL Offs(pOrigin,403.85,100.84,0.00),v60,z0,tPen\WObj:=wPaper;
    MoveL Offs(pOrigin,403.64,101.26,0.00),v40,z0,tPen\WObj:=wPaper;
    MoveL Offs(pOrigin,403.85,100.84,0.00),v40,fine,tPen\WObj:=wPaper;
    MoveL Offs(pOrigin,403.85,100.84,6.00),v60,z5,tPen\WObj:=wPaper;
    MoveL Offs(pOrigin,402.79,102.54,6.00),vTravel,z5,tPen\WObj:=wPaper;
    MoveL Offs(pOrigin,402.79,102.54,0.00),v60,z0,tPen\WObj:=wPaper;
    MoveL Offs(pOrigin,403.00,102.11,0.00),v40,z0,tPen\WObj:=wPaper;
    MoveL Offs(pOrigin,402.79,102.54,0.00),v40,fine,tPen\WObj:=wPaper;
    MoveL Offs(pOrigin,402.79,102.54,6.00),v60,z5,tPen\WObj:=wPaper;
    MoveL Offs(pOrigin,401.94,103.60,6.00),vTravel,z5,tPen\WObj:=wPaper;
    MoveL Offs(pOrigin,401.94,103.60,0.00),v60,z0,tPen\WObj:=wPaper;
    MoveL Offs(pOrigin,402.15,103.18,0.00),v40,z0,tPen\WObj:=wPaper;
    MoveL Offs(pOrigin,401.94,103.60,0.00),v40,z0,tPen\WObj:=wPaper;
    MoveL Offs(pOrigin,401.30,104.24,0.00),v40,z0,tPen\WObj:=wPaper;
    MoveL Offs(pOrigin,401.51,103.81,0.00),v40,z0,tPen\WObj:=wPaper;
    MoveL Offs(pOrigin,401.30,104.24,0.00),v40,z0,tPen\WObj:=wPaper;
    MoveL Offs(pOrigin,400.66,104.88,0.00),v40,z0,tPen\WObj:=wPaper;
    MoveL Offs(pOrigin,400.88,104.45,0.00),v40,z0,tPen\WObj:=wPaper;
    MoveL Offs(pOrigin,400.66,104.88,0.00),v40,z0,tPen\WObj:=wPaper;
    MoveL Offs(pOrigin,400.24,105.09,0.00),v40,z0,tPen\WObj:=wPaper;
    MoveL Offs(pOrigin,400.02,105.51,0.00),v40,z0,tPen\WObj:=wPaper;
    MoveL Offs(pOrigin,400.24,105.09,0.00),v40,fine,tPen\WObj:=wPaper;
    MoveL Offs(pOrigin,400.24,105.09,6.00),v60,z5,tPen\WObj:=wPaper;
    MoveL Offs(pOrigin,398.96,106.36,6.00),vTravel,z5,tPen\WObj:=wPaper;
    MoveL Offs(pOrigin,398.96,106.36,0.00),v60,z0,tPen\WObj:=wPaper;
  ENDPROC

  PROC DrawPart84()
    MoveL Offs(pOrigin,403.14,102.11,0.00),v40,z0,tPen\WObj:=wPaper;
    MoveL Offs(pOrigin,404.56,99.99,0.00),v40,z0,tPen\WObj:=wPaper;
    MoveL Offs(pOrigin,405.83,97.22,0.00),v40,z0,tPen\WObj:=wPaper;
    MoveL Offs(pOrigin,407.04,93.61,0.00),v40,z0,tPen\WObj:=wPaper;
    MoveL Offs(pOrigin,409.80,82.56,0.00),v40,z0,tPen\WObj:=wPaper;
    MoveL Offs(pOrigin,413.62,73.00,0.00),v40,z0,tPen\WObj:=wPaper;
    MoveL Offs(pOrigin,414.40,67.69,0.00),v40,z0,tPen\WObj:=wPaper;
    MoveL Offs(pOrigin,413.84,67.55,0.00),v40,z0,tPen\WObj:=wPaper;
    MoveL Offs(pOrigin,412.77,68.96,0.00),v40,z0,tPen\WObj:=wPaper;
    MoveL Offs(pOrigin,408.52,73.00,0.00),v40,z0,tPen\WObj:=wPaper;
    MoveL Offs(pOrigin,402.36,77.32,0.00),v40,z0,tPen\WObj:=wPaper;
    MoveL Offs(pOrigin,394.71,81.36,0.00),v40,z0,tPen\WObj:=wPaper;
    MoveL Offs(pOrigin,390.46,83.06,0.00),v40,z0,tPen\WObj:=wPaper;
    MoveL Offs(pOrigin,385.36,84.55,0.00),v40,z0,tPen\WObj:=wPaper;
    MoveL Offs(pOrigin,384.94,85.11,0.00),v40,z0,tPen\WObj:=wPaper;
    MoveL Offs(pOrigin,384.94,85.11,0.00),v40,z0,tPen\WObj:=wPaper;
    MoveL Offs(pOrigin,389.61,85.32,0.00),v40,z0,tPen\WObj:=wPaper;
    MoveL Offs(pOrigin,393.65,84.47,0.00),v40,z0,tPen\WObj:=wPaper;
    MoveL Offs(pOrigin,398.33,82.85,0.00),v40,z0,tPen\WObj:=wPaper;
    MoveL Offs(pOrigin,401.09,81.36,0.00),v40,z0,tPen\WObj:=wPaper;
    MoveL Offs(pOrigin,405.34,78.38,0.00),v40,z0,tPen\WObj:=wPaper;
    MoveL Offs(pOrigin,405.98,78.38,0.00),v40,z0,tPen\WObj:=wPaper;
    MoveL Offs(pOrigin,405.90,79.16,0.00),v40,z0,tPen\WObj:=wPaper;
    MoveL Offs(pOrigin,403.21,81.29,0.00),v40,z0,tPen\WObj:=wPaper;
    MoveL Offs(pOrigin,402.36,81.71,0.00),v40,z0,tPen\WObj:=wPaper;
    MoveL Offs(pOrigin,402.65,81.57,0.00),v40,z0,tPen\WObj:=wPaper;
    MoveL Offs(pOrigin,398.33,84.12,0.00),v40,z0,tPen\WObj:=wPaper;
    MoveL Offs(pOrigin,393.86,85.75,0.00),v40,z0,tPen\WObj:=wPaper;
    MoveL Offs(pOrigin,389.61,86.60,0.00),v40,z0,tPen\WObj:=wPaper;
    MoveL Offs(pOrigin,384.73,86.81,0.00),v40,z0,tPen\WObj:=wPaper;
    MoveL Offs(pOrigin,377.50,85.75,0.00),v40,z0,tPen\WObj:=wPaper;
    MoveL Offs(pOrigin,371.12,83.91,0.00),v40,z0,tPen\WObj:=wPaper;
    MoveL Offs(pOrigin,366.02,81.57,0.00),v40,z0,tPen\WObj:=wPaper;
    MoveL Offs(pOrigin,360.92,78.45,0.00),v40,z0,tPen\WObj:=wPaper;
    MoveL Offs(pOrigin,359.01,77.68,0.00),v40,z0,tPen\WObj:=wPaper;
    MoveL Offs(pOrigin,356.04,77.46,0.00),v40,z0,tPen\WObj:=wPaper;
    MoveL Offs(pOrigin,355.40,77.89,0.00),v40,z0,tPen\WObj:=wPaper;
    MoveL Offs(pOrigin,355.40,77.89,0.00),v40,z0,tPen\WObj:=wPaper;
    MoveL Offs(pOrigin,354.55,77.46,0.00),v40,z0,tPen\WObj:=wPaper;
    MoveL Offs(pOrigin,354.20,77.68,0.00),v40,z0,tPen\WObj:=wPaper;
    MoveL Offs(pOrigin,353.70,79.80,0.00),v40,z0,tPen\WObj:=wPaper;
    MoveL Offs(pOrigin,353.06,87.88,0.00),v40,z0,tPen\WObj:=wPaper;
    MoveL Offs(pOrigin,353.27,91.28,0.00),v40,z0,tPen\WObj:=wPaper;
    MoveL Offs(pOrigin,352.42,91.91,0.00),v40,z0,tPen\WObj:=wPaper;
    MoveL Offs(pOrigin,352.00,92.12,0.00),v40,z0,tPen\WObj:=wPaper;
    MoveL Offs(pOrigin,349.38,96.38,0.00),v40,z0,tPen\WObj:=wPaper;
    MoveL Offs(pOrigin,349.02,97.44,0.00),v40,z0,tPen\WObj:=wPaper;
    MoveL Offs(pOrigin,349.17,99.35,0.00),v40,z0,tPen\WObj:=wPaper;
    MoveL Offs(pOrigin,350.73,101.69,0.00),v40,z0,tPen\WObj:=wPaper;
    MoveL Offs(pOrigin,357.10,107.78,0.00),v40,z0,tPen\WObj:=wPaper;
    MoveL Offs(pOrigin,358.30,108.35,0.00),v40,z0,tPen\WObj:=wPaper;
    MoveL Offs(pOrigin,358.80,109.27,0.00),v40,z0,tPen\WObj:=wPaper;
    MoveL Offs(pOrigin,366.02,113.66,0.00),v40,z0,tPen\WObj:=wPaper;
    MoveL Offs(pOrigin,377.29,119.40,0.00),v40,z0,tPen\WObj:=wPaper;
    MoveL Offs(pOrigin,384.94,122.58,0.00),v40,z0,tPen\WObj:=wPaper;
    MoveL Offs(pOrigin,387.49,123.36,0.00),v40,z0,tPen\WObj:=wPaper;
    MoveL Offs(pOrigin,388.55,123.36,0.00),v40,fine,tPen\WObj:=wPaper;
    MoveL Offs(pOrigin,388.55,123.36,6.00),v60,z5,tPen\WObj:=wPaper;
    MoveL Offs(pOrigin,384.51,125.70,6.00),vTravel,z5,tPen\WObj:=wPaper;
    MoveL Offs(pOrigin,384.51,125.70,0.00),v60,z0,tPen\WObj:=wPaper;
    MoveL Offs(pOrigin,384.94,126.27,0.00),v40,z0,tPen\WObj:=wPaper;
    MoveL Offs(pOrigin,390.04,127.82,0.00),v40,z0,tPen\WObj:=wPaper;
    MoveL Offs(pOrigin,389.19,132.07,0.00),v40,z0,tPen\WObj:=wPaper;
    MoveL Offs(pOrigin,389.19,136.96,0.00),v40,z0,tPen\WObj:=wPaper;
    MoveL Offs(pOrigin,388.41,140.15,0.00),v40,z0,tPen\WObj:=wPaper;
    MoveL Offs(pOrigin,385.36,143.41,0.00),v40,z0,tPen\WObj:=wPaper;
    MoveL Offs(pOrigin,384.09,142.91,0.00),v40,z0,tPen\WObj:=wPaper;
    MoveL Offs(pOrigin,378.77,138.95,0.00),v40,z0,tPen\WObj:=wPaper;
    MoveL Offs(pOrigin,378.00,138.88,0.00),v40,z0,tPen\WObj:=wPaper;
    MoveL Offs(pOrigin,378.35,139.73,0.00),v40,z0,tPen\WObj:=wPaper;
    MoveL Offs(pOrigin,384.30,144.82,0.00),v40,z0,tPen\WObj:=wPaper;
    MoveL Offs(pOrigin,385.08,145.89,0.00),v40,z0,tPen\WObj:=wPaper;
    MoveL Offs(pOrigin,385.58,147.38,0.00),v40,z0,tPen\WObj:=wPaper;
    MoveL Offs(pOrigin,385.58,148.86,0.00),v40,z0,tPen\WObj:=wPaper;
    MoveL Offs(pOrigin,385.01,150.77,0.00),v40,z0,tPen\WObj:=wPaper;
    MoveL Offs(pOrigin,380.62,160.34,0.00),v40,z0,tPen\WObj:=wPaper;
    MoveL Offs(pOrigin,379.41,163.74,0.00),v40,z0,tPen\WObj:=wPaper;
    MoveL Offs(pOrigin,378.99,163.88,0.00),v40,z0,tPen\WObj:=wPaper;
    MoveL Offs(pOrigin,378.49,163.52,0.00),v40,z0,tPen\WObj:=wPaper;
    MoveL Offs(pOrigin,366.45,148.86,0.00),v40,z0,tPen\WObj:=wPaper;
    MoveL Offs(pOrigin,365.81,148.65,0.00),v40,z0,tPen\WObj:=wPaper;
    MoveL Offs(pOrigin,365.81,148.65,0.00),v40,z0,tPen\WObj:=wPaper;
    MoveL Offs(pOrigin,365.74,147.80,0.00),v40,z0,tPen\WObj:=wPaper;
    MoveL Offs(pOrigin,364.54,147.16,0.00),v40,z0,tPen\WObj:=wPaper;
    MoveL Offs(pOrigin,359.01,140.36,0.00),v40,fine,tPen\WObj:=wPaper;
    MoveL Offs(pOrigin,359.01,140.36,6.00),v60,z5,tPen\WObj:=wPaper;
    MoveL Offs(pOrigin,360.08,138.45,6.00),vTravel,z5,tPen\WObj:=wPaper;
    MoveL Offs(pOrigin,360.08,138.45,0.00),v60,z0,tPen\WObj:=wPaper;
    MoveL Offs(pOrigin,358.80,137.39,0.00),v40,z0,tPen\WObj:=wPaper;
    MoveL Offs(pOrigin,358.59,136.75,0.00),v40,z0,tPen\WObj:=wPaper;
    MoveL Offs(pOrigin,358.59,136.75,0.00),v40,z0,tPen\WObj:=wPaper;
    MoveL Offs(pOrigin,357.95,136.32,0.00),v40,z0,tPen\WObj:=wPaper;
    MoveL Offs(pOrigin,355.90,133.56,0.00),v40,z0,tPen\WObj:=wPaper;
    MoveL Offs(pOrigin,355.61,132.50,0.00),v40,z0,tPen\WObj:=wPaper;
    MoveL Offs(pOrigin,355.61,132.50,0.00),v40,z0,tPen\WObj:=wPaper;
    MoveL Offs(pOrigin,356.67,132.93,0.00),v40,z0,tPen\WObj:=wPaper;
    MoveL Offs(pOrigin,358.94,135.90,0.00),v40,z0,tPen\WObj:=wPaper;
    MoveL Offs(pOrigin,359.01,136.54,0.00),v40,z0,tPen\WObj:=wPaper;
    MoveL Offs(pOrigin,359.01,136.54,0.00),v40,z0,tPen\WObj:=wPaper;
    MoveL Offs(pOrigin,359.65,136.54,0.00),v40,z0,tPen\WObj:=wPaper;
    MoveL Offs(pOrigin,360.50,137.39,0.00),v40,z0,tPen\WObj:=wPaper;
    MoveL Offs(pOrigin,360.50,138.24,0.00),v40,z0,tPen\WObj:=wPaper;
    MoveL Offs(pOrigin,360.50,138.24,0.00),v40,z0,tPen\WObj:=wPaper;
    MoveL Offs(pOrigin,360.92,138.24,0.00),v40,z0,tPen\WObj:=wPaper;
    MoveL Offs(pOrigin,361.99,139.30,0.00),v40,z0,tPen\WObj:=wPaper;
    MoveL Offs(pOrigin,362.20,140.15,0.00),v40,z0,tPen\WObj:=wPaper;
    MoveL Offs(pOrigin,362.20,140.15,0.00),v40,z0,tPen\WObj:=wPaper;
    MoveL Offs(pOrigin,363.26,141.21,0.00),v40,z0,tPen\WObj:=wPaper;
    MoveL Offs(pOrigin,363.26,141.21,0.00),v40,z0,tPen\WObj:=wPaper;
    MoveL Offs(pOrigin,364.54,141.64,0.00),v40,z0,tPen\WObj:=wPaper;
    MoveL Offs(pOrigin,366.02,143.76,0.00),v40,z0,tPen\WObj:=wPaper;
    MoveL Offs(pOrigin,369.64,146.95,0.00),v40,z0,tPen\WObj:=wPaper;
    MoveL Offs(pOrigin,375.16,150.77,0.00),v40,fine,tPen\WObj:=wPaper;
    MoveL Offs(pOrigin,375.16,150.77,6.00),v60,z5,tPen\WObj:=wPaper;
    MoveL Offs(pOrigin,371.98,155.24,6.00),vTravel,z5,tPen\WObj:=wPaper;
    MoveL Offs(pOrigin,371.98,155.24,0.00),v60,z0,tPen\WObj:=wPaper;
    MoveL Offs(pOrigin,372.83,156.09,0.00),v40,z0,tPen\WObj:=wPaper;
    MoveL Offs(pOrigin,371.98,155.24,0.00),v40,fine,tPen\WObj:=wPaper;
    MoveL Offs(pOrigin,371.98,155.24,6.00),v60,z5,tPen\WObj:=wPaper;
    MoveL Offs(pOrigin,373.04,156.30,6.00),vTravel,z5,tPen\WObj:=wPaper;
  ENDPROC

  PROC DrawPart85()
    MoveL Offs(pOrigin,373.04,156.30,0.00),v60,z0,tPen\WObj:=wPaper;
    MoveL Offs(pOrigin,373.89,157.36,0.00),v40,z0,tPen\WObj:=wPaper;
    MoveL Offs(pOrigin,373.04,156.30,0.00),v40,fine,tPen\WObj:=wPaper;
    MoveL Offs(pOrigin,373.04,156.30,6.00),v60,z5,tPen\WObj:=wPaper;
    MoveL Offs(pOrigin,372.40,158.00,6.00),vTravel,z5,tPen\WObj:=wPaper;
    MoveL Offs(pOrigin,372.40,158.00,0.00),v60,z0,tPen\WObj:=wPaper;
    MoveL Offs(pOrigin,372.61,158.43,0.00),v40,z0,tPen\WObj:=wPaper;
    MoveL Offs(pOrigin,372.40,158.00,0.00),v40,fine,tPen\WObj:=wPaper;
    MoveL Offs(pOrigin,372.40,158.00,6.00),v60,z5,tPen\WObj:=wPaper;
    MoveL Offs(pOrigin,373.25,159.06,6.00),vTravel,z5,tPen\WObj:=wPaper;
    MoveL Offs(pOrigin,373.25,159.06,0.00),v60,z0,tPen\WObj:=wPaper;
    MoveL Offs(pOrigin,373.46,159.49,0.00),v40,z0,tPen\WObj:=wPaper;
    MoveL Offs(pOrigin,373.25,159.06,0.00),v40,fine,tPen\WObj:=wPaper;
    MoveL Offs(pOrigin,373.25,159.06,6.00),v60,z5,tPen\WObj:=wPaper;
    MoveL Offs(pOrigin,374.31,158.00,6.00),vTravel,z5,tPen\WObj:=wPaper;
    MoveL Offs(pOrigin,374.31,158.00,0.00),v60,z0,tPen\WObj:=wPaper;
    MoveL Offs(pOrigin,374.74,158.43,0.00),v40,z0,tPen\WObj:=wPaper;
    MoveL Offs(pOrigin,374.31,158.00,0.00),v40,fine,tPen\WObj:=wPaper;
    MoveL Offs(pOrigin,374.31,158.00,6.00),v60,z5,tPen\WObj:=wPaper;
    MoveL Offs(pOrigin,375.16,159.06,6.00),vTravel,z5,tPen\WObj:=wPaper;
    MoveL Offs(pOrigin,375.16,159.06,0.00),v60,z0,tPen\WObj:=wPaper;
    MoveL Offs(pOrigin,375.80,159.70,0.00),v40,z0,tPen\WObj:=wPaper;
    MoveL Offs(pOrigin,375.16,159.06,0.00),v40,fine,tPen\WObj:=wPaper;
    MoveL Offs(pOrigin,375.16,159.06,6.00),v60,z5,tPen\WObj:=wPaper;
    MoveL Offs(pOrigin,376.01,160.12,6.00),vTravel,z5,tPen\WObj:=wPaper;
    MoveL Offs(pOrigin,376.01,160.12,0.00),v60,z0,tPen\WObj:=wPaper;
    MoveL Offs(pOrigin,376.65,160.76,0.00),v40,z0,tPen\WObj:=wPaper;
    MoveL Offs(pOrigin,376.01,160.12,0.00),v40,fine,tPen\WObj:=wPaper;
    MoveL Offs(pOrigin,376.01,160.12,6.00),v60,z5,tPen\WObj:=wPaper;
    MoveL Offs(pOrigin,377.50,162.04,6.00),vTravel,z5,tPen\WObj:=wPaper;
    MoveL Offs(pOrigin,377.50,162.04,0.00),v60,z0,tPen\WObj:=wPaper;
    MoveL Offs(pOrigin,377.92,162.46,0.00),v40,z0,tPen\WObj:=wPaper;
    MoveL Offs(pOrigin,377.50,162.04,0.00),v40,fine,tPen\WObj:=wPaper;
    MoveL Offs(pOrigin,377.50,162.04,6.00),v60,z5,tPen\WObj:=wPaper;
    MoveL Offs(pOrigin,376.23,163.10,6.00),vTravel,z5,tPen\WObj:=wPaper;
    MoveL Offs(pOrigin,376.23,163.10,0.00),v60,z0,tPen\WObj:=wPaper;
    MoveL Offs(pOrigin,376.65,163.52,0.00),v40,z0,tPen\WObj:=wPaper;
    MoveL Offs(pOrigin,376.23,163.10,0.00),v40,z0,tPen\WObj:=wPaper;
    MoveL Offs(pOrigin,376.86,163.95,0.00),v40,z0,tPen\WObj:=wPaper;
    MoveL Offs(pOrigin,377.29,164.38,0.00),v40,z0,tPen\WObj:=wPaper;
    MoveL Offs(pOrigin,376.86,163.95,0.00),v40,fine,tPen\WObj:=wPaper;
    MoveL Offs(pOrigin,376.86,163.95,6.00),v60,z5,tPen\WObj:=wPaper;
    MoveL Offs(pOrigin,378.77,166.71,6.00),vTravel,z5,tPen\WObj:=wPaper;
    MoveL Offs(pOrigin,378.77,166.71,0.00),v60,z0,tPen\WObj:=wPaper;
    MoveL Offs(pOrigin,378.99,167.14,0.00),v40,z0,tPen\WObj:=wPaper;
    MoveL Offs(pOrigin,378.77,166.71,0.00),v40,fine,tPen\WObj:=wPaper;
    MoveL Offs(pOrigin,378.77,166.71,6.00),v60,z5,tPen\WObj:=wPaper;
    MoveL Offs(pOrigin,373.67,169.69,6.00),vTravel,z5,tPen\WObj:=wPaper;
    MoveL Offs(pOrigin,373.67,169.69,0.00),v60,z0,tPen\WObj:=wPaper;
    MoveL Offs(pOrigin,374.10,170.32,0.00),v40,z0,tPen\WObj:=wPaper;
    MoveL Offs(pOrigin,373.67,169.69,0.00),v40,fine,tPen\WObj:=wPaper;
    MoveL Offs(pOrigin,373.67,169.69,6.00),v60,z5,tPen\WObj:=wPaper;
    MoveL Offs(pOrigin,369.85,171.18,6.00),vTravel,z5,tPen\WObj:=wPaper;
    MoveL Offs(pOrigin,369.85,171.18,0.00),v60,z0,tPen\WObj:=wPaper;
    MoveL Offs(pOrigin,369.85,172.24,0.00),v40,z0,tPen\WObj:=wPaper;
    MoveL Offs(pOrigin,371.27,176.06,0.00),v40,z0,tPen\WObj:=wPaper;
    MoveL Offs(pOrigin,375.38,184.99,0.00),v40,z0,tPen\WObj:=wPaper;
    MoveL Offs(pOrigin,375.38,184.99,0.00),v40,z0,tPen\WObj:=wPaper;
    MoveL Offs(pOrigin,375.59,186.69,0.00),v40,z0,tPen\WObj:=wPaper;
    MoveL Offs(pOrigin,374.95,187.75,0.00),v40,z0,tPen\WObj:=wPaper;
    MoveL Offs(pOrigin,375.38,186.90,0.00),v40,z0,tPen\WObj:=wPaper;
    MoveL Offs(pOrigin,375.16,187.32,0.00),v40,z0,tPen\WObj:=wPaper;
    MoveL Offs(pOrigin,375.38,186.90,0.00),v40,fine,tPen\WObj:=wPaper;
    MoveL Offs(pOrigin,375.38,186.90,6.00),v60,z5,tPen\WObj:=wPaper;
    MoveL Offs(pOrigin,376.44,188.18,6.00),vTravel,z5,tPen\WObj:=wPaper;
    MoveL Offs(pOrigin,376.44,188.18,0.00),v60,z0,tPen\WObj:=wPaper;
    MoveL Offs(pOrigin,375.38,189.24,0.00),v40,z0,tPen\WObj:=wPaper;
    MoveL Offs(pOrigin,376.44,188.18,0.00),v40,fine,tPen\WObj:=wPaper;
    MoveL Offs(pOrigin,376.44,188.18,6.00),v60,z5,tPen\WObj:=wPaper;
    MoveL Offs(pOrigin,377.08,187.11,6.00),vTravel,z5,tPen\WObj:=wPaper;
    MoveL Offs(pOrigin,377.08,187.11,0.00),v60,z0,tPen\WObj:=wPaper;
    MoveL Offs(pOrigin,376.65,187.75,0.00),v40,z0,tPen\WObj:=wPaper;
    MoveL Offs(pOrigin,377.08,187.11,0.00),v40,fine,tPen\WObj:=wPaper;
    MoveL Offs(pOrigin,377.08,187.11,6.00),v60,z5,tPen\WObj:=wPaper;
    MoveL Offs(pOrigin,378.99,186.90,6.00),vTravel,z5,tPen\WObj:=wPaper;
    MoveL Offs(pOrigin,378.99,186.90,0.00),v60,z0,tPen\WObj:=wPaper;
    MoveL Offs(pOrigin,378.77,185.62,0.00),v40,fine,tPen\WObj:=wPaper;
    MoveL Offs(pOrigin,378.77,185.62,6.00),v60,z5,tPen\WObj:=wPaper;
    MoveL Offs(pOrigin,375.38,184.99,6.00),vTravel,z5,tPen\WObj:=wPaper;
    MoveL Offs(pOrigin,375.38,184.99,0.00),v60,z0,tPen\WObj:=wPaper;
    MoveL Offs(pOrigin,376.23,184.92,0.00),v40,z0,tPen\WObj:=wPaper;
    MoveL Offs(pOrigin,376.65,184.14,0.00),v40,z0,tPen\WObj:=wPaper;
    MoveL Offs(pOrigin,378.14,176.70,0.00),v40,z0,tPen\WObj:=wPaper;
    MoveL Offs(pOrigin,380.05,171.60,0.00),v40,z0,tPen\WObj:=wPaper;
    MoveL Offs(pOrigin,380.05,169.48,0.00),v40,z0,tPen\WObj:=wPaper;
    MoveL Offs(pOrigin,378.85,166.50,0.00),v40,z0,tPen\WObj:=wPaper;
    MoveL Offs(pOrigin,377.29,164.16,0.00),v40,z0,tPen\WObj:=wPaper;
    MoveL Offs(pOrigin,365.39,148.86,0.00),v40,z0,tPen\WObj:=wPaper;
    MoveL Offs(pOrigin,365.39,148.86,0.00),v40,z0,tPen\WObj:=wPaper;
    MoveL Offs(pOrigin,364.75,148.23,0.00),v40,z0,tPen\WObj:=wPaper;
    MoveL Offs(pOrigin,364.54,147.38,0.00),v40,fine,tPen\WObj:=wPaper;
    MoveL Offs(pOrigin,364.54,147.38,6.00),v60,z5,tPen\WObj:=wPaper;
    MoveL Offs(pOrigin,365.60,149.50,6.00),vTravel,z5,tPen\WObj:=wPaper;
    MoveL Offs(pOrigin,365.60,149.50,0.00),v60,z0,tPen\WObj:=wPaper;
    MoveL Offs(pOrigin,366.02,149.93,0.00),v40,z0,tPen\WObj:=wPaper;
    MoveL Offs(pOrigin,365.60,149.50,0.00),v40,fine,tPen\WObj:=wPaper;
    MoveL Offs(pOrigin,365.60,149.50,6.00),v60,z5,tPen\WObj:=wPaper;
    MoveL Offs(pOrigin,367.30,149.50,6.00),vTravel,z5,tPen\WObj:=wPaper;
    MoveL Offs(pOrigin,367.30,149.50,0.00),v60,z0,tPen\WObj:=wPaper;
    MoveL Offs(pOrigin,367.51,149.93,0.00),v40,z0,tPen\WObj:=wPaper;
    MoveL Offs(pOrigin,367.30,149.50,0.00),v40,fine,tPen\WObj:=wPaper;
    MoveL Offs(pOrigin,367.30,149.50,6.00),v60,z5,tPen\WObj:=wPaper;
    MoveL Offs(pOrigin,368.15,150.56,6.00),vTravel,z5,tPen\WObj:=wPaper;
    MoveL Offs(pOrigin,368.15,150.56,0.00),v60,z0,tPen\WObj:=wPaper;
    MoveL Offs(pOrigin,368.58,150.99,0.00),v40,z0,tPen\WObj:=wPaper;
    MoveL Offs(pOrigin,368.15,150.56,0.00),v40,z0,tPen\WObj:=wPaper;
    MoveL Offs(pOrigin,368.79,151.41,0.00),v40,z0,tPen\WObj:=wPaper;
    MoveL Offs(pOrigin,369.64,152.26,0.00),v40,z0,tPen\WObj:=wPaper;
    MoveL Offs(pOrigin,368.79,151.41,0.00),v40,fine,tPen\WObj:=wPaper;
    MoveL Offs(pOrigin,368.79,151.41,6.00),v60,z5,tPen\WObj:=wPaper;
    MoveL Offs(pOrigin,367.94,152.48,6.00),vTravel,z5,tPen\WObj:=wPaper;
    MoveL Offs(pOrigin,367.94,152.48,0.00),v60,z0,tPen\WObj:=wPaper;
    MoveL Offs(pOrigin,368.36,152.90,0.00),v40,z0,tPen\WObj:=wPaper;
    MoveL Offs(pOrigin,367.94,152.48,0.00),v40,fine,tPen\WObj:=wPaper;
    MoveL Offs(pOrigin,367.94,152.48,6.00),v60,z5,tPen\WObj:=wPaper;
    MoveL Offs(pOrigin,367.09,151.41,6.00),vTravel,z5,tPen\WObj:=wPaper;
    MoveL Offs(pOrigin,367.09,151.41,0.00),v60,z0,tPen\WObj:=wPaper;
    MoveL Offs(pOrigin,367.51,151.84,0.00),v40,z0,tPen\WObj:=wPaper;
    MoveL Offs(pOrigin,367.09,151.41,0.00),v40,fine,tPen\WObj:=wPaper;
    MoveL Offs(pOrigin,367.09,151.41,6.00),v60,z5,tPen\WObj:=wPaper;
  ENDPROC

  PROC DrawPart86()
    MoveL Offs(pOrigin,368.79,153.54,6.00),vTravel,z5,tPen\WObj:=wPaper;
    MoveL Offs(pOrigin,368.79,153.54,0.00),v60,z0,tPen\WObj:=wPaper;
    MoveL Offs(pOrigin,369.21,153.96,0.00),v40,z0,tPen\WObj:=wPaper;
    MoveL Offs(pOrigin,368.79,153.54,0.00),v40,fine,tPen\WObj:=wPaper;
    MoveL Offs(pOrigin,368.79,153.54,6.00),v60,z5,tPen\WObj:=wPaper;
    MoveL Offs(pOrigin,370.06,155.24,6.00),vTravel,z5,tPen\WObj:=wPaper;
    MoveL Offs(pOrigin,370.06,155.24,0.00),v60,z0,tPen\WObj:=wPaper;
    MoveL Offs(pOrigin,370.70,155.88,0.00),v40,z0,tPen\WObj:=wPaper;
    MoveL Offs(pOrigin,370.06,155.24,0.00),v40,fine,tPen\WObj:=wPaper;
    MoveL Offs(pOrigin,370.06,155.24,6.00),v60,z5,tPen\WObj:=wPaper;
    MoveL Offs(pOrigin,371.12,156.51,6.00),vTravel,z5,tPen\WObj:=wPaper;
    MoveL Offs(pOrigin,371.12,156.51,0.00),v60,z0,tPen\WObj:=wPaper;
    MoveL Offs(pOrigin,371.55,156.94,0.00),v40,z0,tPen\WObj:=wPaper;
    MoveL Offs(pOrigin,371.12,156.51,0.00),v40,fine,tPen\WObj:=wPaper;
    MoveL Offs(pOrigin,371.12,156.51,6.00),v60,z5,tPen\WObj:=wPaper;
    MoveL Offs(pOrigin,366.45,157.79,6.00),vTravel,z5,tPen\WObj:=wPaper;
    MoveL Offs(pOrigin,366.45,157.79,0.00),v60,z0,tPen\WObj:=wPaper;
    MoveL Offs(pOrigin,366.66,158.21,0.00),v40,z0,tPen\WObj:=wPaper;
    MoveL Offs(pOrigin,366.45,157.79,0.00),v40,fine,tPen\WObj:=wPaper;
    MoveL Offs(pOrigin,366.45,157.79,6.00),v60,z5,tPen\WObj:=wPaper;
    MoveL Offs(pOrigin,364.96,155.02,6.00),vTravel,z5,tPen\WObj:=wPaper;
    MoveL Offs(pOrigin,364.96,155.02,0.00),v60,z0,tPen\WObj:=wPaper;
    MoveL Offs(pOrigin,365.17,155.45,0.00),v40,z0,tPen\WObj:=wPaper;
    MoveL Offs(pOrigin,364.96,155.02,0.00),v40,fine,tPen\WObj:=wPaper;
    MoveL Offs(pOrigin,364.96,155.02,6.00),v60,z5,tPen\WObj:=wPaper;
    MoveL Offs(pOrigin,361.99,148.86,6.00),vTravel,z5,tPen\WObj:=wPaper;
    MoveL Offs(pOrigin,361.99,148.86,0.00),v60,z0,tPen\WObj:=wPaper;
    MoveL Offs(pOrigin,368.29,160.98,0.00),v40,z0,tPen\WObj:=wPaper;
    MoveL Offs(pOrigin,376.86,174.36,0.00),v40,fine,tPen\WObj:=wPaper;
    MoveL Offs(pOrigin,376.86,174.36,6.00),v60,z5,tPen\WObj:=wPaper;
    MoveL Offs(pOrigin,374.10,188.18,6.00),vTravel,z5,tPen\WObj:=wPaper;
    MoveL Offs(pOrigin,374.10,188.18,0.00),v60,z0,tPen\WObj:=wPaper;
    MoveL Offs(pOrigin,374.38,188.03,0.00),v40,z0,tPen\WObj:=wPaper;
    MoveL Offs(pOrigin,372.40,189.02,0.00),v40,z0,tPen\WObj:=wPaper;
    MoveL Offs(pOrigin,371.34,189.02,0.00),v40,z0,tPen\WObj:=wPaper;
    MoveL Offs(pOrigin,370.27,188.18,0.00),v40,z0,tPen\WObj:=wPaper;
    MoveL Offs(pOrigin,368.43,184.99,0.00),v40,z0,tPen\WObj:=wPaper;
    MoveL Offs(pOrigin,365.95,178.61,0.00),v40,z0,tPen\WObj:=wPaper;
    MoveL Offs(pOrigin,362.62,167.77,0.00),v40,z0,tPen\WObj:=wPaper;
    MoveL Offs(pOrigin,357.74,149.50,0.00),v40,z0,tPen\WObj:=wPaper;
    MoveL Offs(pOrigin,353.70,131.86,0.00),v40,z0,tPen\WObj:=wPaper;
    MoveL Offs(pOrigin,354.12,130.80,0.00),v40,z0,tPen\WObj:=wPaper;
    MoveL Offs(pOrigin,353.91,130.38,0.00),v40,z0,tPen\WObj:=wPaper;
    MoveL Offs(pOrigin,354.12,130.80,0.00),v40,z0,tPen\WObj:=wPaper;
    MoveL Offs(pOrigin,353.91,130.38,0.00),v40,fine,tPen\WObj:=wPaper;
    MoveL Offs(pOrigin,353.91,130.38,6.00),v60,z5,tPen\WObj:=wPaper;
    MoveL Offs(pOrigin,355.61,128.68,6.00),vTravel,z5,tPen\WObj:=wPaper;
    MoveL Offs(pOrigin,355.61,128.68,0.00),v60,z0,tPen\WObj:=wPaper;
    MoveL Offs(pOrigin,356.04,129.31,0.00),v40,z0,tPen\WObj:=wPaper;
    MoveL Offs(pOrigin,355.61,128.68,0.00),v40,fine,tPen\WObj:=wPaper;
    MoveL Offs(pOrigin,355.61,128.68,6.00),v60,z5,tPen\WObj:=wPaper;
    MoveL Offs(pOrigin,356.67,128.04,6.00),vTravel,z5,tPen\WObj:=wPaper;
    MoveL Offs(pOrigin,356.67,128.04,0.00),v60,z0,tPen\WObj:=wPaper;
    MoveL Offs(pOrigin,357.31,128.89,0.00),v40,z0,tPen\WObj:=wPaper;
    MoveL Offs(pOrigin,356.67,128.04,0.00),v40,z0,tPen\WObj:=wPaper;
    MoveL Offs(pOrigin,356.25,127.40,0.00),v40,z0,tPen\WObj:=wPaper;
    MoveL Offs(pOrigin,356.46,127.82,0.00),v40,z0,tPen\WObj:=wPaper;
    MoveL Offs(pOrigin,356.25,127.40,0.00),v40,fine,tPen\WObj:=wPaper;
    MoveL Offs(pOrigin,356.25,127.40,6.00),v60,z5,tPen\WObj:=wPaper;
    MoveL Offs(pOrigin,355.61,126.34,6.00),vTravel,z5,tPen\WObj:=wPaper;
    MoveL Offs(pOrigin,355.61,126.34,0.00),v60,z0,tPen\WObj:=wPaper;
    MoveL Offs(pOrigin,355.83,126.76,0.00),v40,z0,tPen\WObj:=wPaper;
    MoveL Offs(pOrigin,355.61,126.34,0.00),v40,fine,tPen\WObj:=wPaper;
    MoveL Offs(pOrigin,355.61,126.34,6.00),v60,z5,tPen\WObj:=wPaper;
    MoveL Offs(pOrigin,353.70,125.70,6.00),vTravel,z5,tPen\WObj:=wPaper;
    MoveL Offs(pOrigin,353.70,125.70,0.00),v60,z0,tPen\WObj:=wPaper;
    MoveL Offs(pOrigin,354.12,126.34,0.00),v40,z0,tPen\WObj:=wPaper;
    MoveL Offs(pOrigin,353.70,125.70,0.00),v40,z0,tPen\WObj:=wPaper;
    MoveL Offs(pOrigin,352.85,125.06,0.00),v40,z0,tPen\WObj:=wPaper;
    MoveL Offs(pOrigin,352.64,125.70,0.00),v40,z0,tPen\WObj:=wPaper;
    MoveL Offs(pOrigin,353.70,128.25,0.00),v40,z0,tPen\WObj:=wPaper;
    MoveL Offs(pOrigin,354.05,130.38,0.00),v40,z0,tPen\WObj:=wPaper;
    MoveL Offs(pOrigin,354.98,131.23,0.00),v40,z0,tPen\WObj:=wPaper;
    MoveL Offs(pOrigin,355.61,132.50,0.00),v40,fine,tPen\WObj:=wPaper;
    MoveL Offs(pOrigin,355.61,132.50,6.00),v60,z5,tPen\WObj:=wPaper;
    MoveL Offs(pOrigin,358.38,130.38,6.00),vTravel,z5,tPen\WObj:=wPaper;
    MoveL Offs(pOrigin,358.38,130.38,0.00),v60,z0,tPen\WObj:=wPaper;
    MoveL Offs(pOrigin,358.80,130.80,0.00),v40,z0,tPen\WObj:=wPaper;
    MoveL Offs(pOrigin,358.38,130.38,0.00),v40,fine,tPen\WObj:=wPaper;
    MoveL Offs(pOrigin,358.38,130.38,6.00),v60,z5,tPen\WObj:=wPaper;
    MoveL Offs(pOrigin,359.23,131.44,6.00),vTravel,z5,tPen\WObj:=wPaper;
    MoveL Offs(pOrigin,359.23,131.44,0.00),v60,z0,tPen\WObj:=wPaper;
    MoveL Offs(pOrigin,359.65,131.86,0.00),v40,z0,tPen\WObj:=wPaper;
    MoveL Offs(pOrigin,359.23,131.44,0.00),v40,fine,tPen\WObj:=wPaper;
    MoveL Offs(pOrigin,359.23,131.44,6.00),v60,z5,tPen\WObj:=wPaper;
    MoveL Offs(pOrigin,360.08,132.50,6.00),vTravel,z5,tPen\WObj:=wPaper;
    MoveL Offs(pOrigin,360.08,132.50,0.00),v60,z0,tPen\WObj:=wPaper;
    MoveL Offs(pOrigin,364.75,137.18,0.00),v40,z0,tPen\WObj:=wPaper;
    MoveL Offs(pOrigin,360.08,132.50,0.00),v40,fine,tPen\WObj:=wPaper;
    MoveL Offs(pOrigin,360.08,132.50,6.00),v60,z5,tPen\WObj:=wPaper;
    MoveL Offs(pOrigin,359.23,133.35,6.00),vTravel,z5,tPen\WObj:=wPaper;
    MoveL Offs(pOrigin,359.23,133.35,0.00),v60,z0,tPen\WObj:=wPaper;
    MoveL Offs(pOrigin,360.08,134.20,0.00),v40,z0,tPen\WObj:=wPaper;
    MoveL Offs(pOrigin,359.23,133.35,0.00),v40,fine,tPen\WObj:=wPaper;
    MoveL Offs(pOrigin,359.23,133.35,6.00),v60,z5,tPen\WObj:=wPaper;
    MoveL Offs(pOrigin,360.29,134.41,6.00),vTravel,z5,tPen\WObj:=wPaper;
    MoveL Offs(pOrigin,360.29,134.41,0.00),v60,z0,tPen\WObj:=wPaper;
    MoveL Offs(pOrigin,360.71,134.84,0.00),v40,z0,tPen\WObj:=wPaper;
    MoveL Offs(pOrigin,360.29,134.41,0.00),v40,fine,tPen\WObj:=wPaper;
    MoveL Offs(pOrigin,360.29,134.41,6.00),v60,z5,tPen\WObj:=wPaper;
    MoveL Offs(pOrigin,361.77,135.90,6.00),vTravel,z5,tPen\WObj:=wPaper;
    MoveL Offs(pOrigin,361.77,135.90,0.00),v60,z0,tPen\WObj:=wPaper;
    MoveL Offs(pOrigin,362.62,136.75,0.00),v40,z0,tPen\WObj:=wPaper;
    MoveL Offs(pOrigin,361.77,135.90,0.00),v40,fine,tPen\WObj:=wPaper;
    MoveL Offs(pOrigin,361.77,135.90,6.00),v60,z5,tPen\WObj:=wPaper;
    MoveL Offs(pOrigin,363.48,137.39,6.00),vTravel,z5,tPen\WObj:=wPaper;
    MoveL Offs(pOrigin,363.48,137.39,0.00),v60,z0,tPen\WObj:=wPaper;
    MoveL Offs(pOrigin,363.90,137.81,0.00),v40,z0,tPen\WObj:=wPaper;
    MoveL Offs(pOrigin,363.48,137.39,0.00),v40,fine,tPen\WObj:=wPaper;
    MoveL Offs(pOrigin,363.48,137.39,6.00),v60,z5,tPen\WObj:=wPaper;
    MoveL Offs(pOrigin,365.39,138.88,6.00),vTravel,z5,tPen\WObj:=wPaper;
    MoveL Offs(pOrigin,365.39,138.88,0.00),v60,z0,tPen\WObj:=wPaper;
    MoveL Offs(pOrigin,365.81,139.30,0.00),v40,z0,tPen\WObj:=wPaper;
    MoveL Offs(pOrigin,365.39,138.88,0.00),v40,fine,tPen\WObj:=wPaper;
    MoveL Offs(pOrigin,365.39,138.88,6.00),v60,z5,tPen\WObj:=wPaper;
    MoveL Offs(pOrigin,367.09,138.88,6.00),vTravel,z5,tPen\WObj:=wPaper;
    MoveL Offs(pOrigin,367.09,138.88,0.00),v60,z0,tPen\WObj:=wPaper;
    MoveL Offs(pOrigin,367.51,139.30,0.00),v40,z0,tPen\WObj:=wPaper;
    MoveL Offs(pOrigin,367.09,138.88,0.00),v40,fine,tPen\WObj:=wPaper;
    MoveL Offs(pOrigin,367.09,138.88,6.00),v60,z5,tPen\WObj:=wPaper;
  ENDPROC

  PROC DrawPart87()
    MoveL Offs(pOrigin,364.33,141.64,6.00),vTravel,z5,tPen\WObj:=wPaper;
    MoveL Offs(pOrigin,364.33,141.64,0.00),v60,z0,tPen\WObj:=wPaper;
    MoveL Offs(pOrigin,365.17,142.49,0.00),v40,z0,tPen\WObj:=wPaper;
    MoveL Offs(pOrigin,364.33,141.64,0.00),v40,z0,tPen\WObj:=wPaper;
    MoveL Offs(pOrigin,363.26,141.21,0.00),v40,z0,tPen\WObj:=wPaper;
    MoveL Offs(pOrigin,363.33,141.85,0.00),v40,z0,tPen\WObj:=wPaper;
    MoveL Offs(pOrigin,365.17,143.62,0.00),v40,z0,tPen\WObj:=wPaper;
    MoveL Offs(pOrigin,365.81,143.76,0.00),v40,z0,tPen\WObj:=wPaper;
    MoveL Offs(pOrigin,365.81,143.76,0.00),v40,z0,tPen\WObj:=wPaper;
    MoveL Offs(pOrigin,366.88,144.82,0.00),v40,z0,tPen\WObj:=wPaper;
    MoveL Offs(pOrigin,367.73,145.46,0.00),v40,z0,tPen\WObj:=wPaper;
    MoveL Offs(pOrigin,368.15,145.89,0.00),v40,z0,tPen\WObj:=wPaper;
    MoveL Offs(pOrigin,367.73,145.46,0.00),v40,fine,tPen\WObj:=wPaper;
    MoveL Offs(pOrigin,367.73,145.46,6.00),v60,z5,tPen\WObj:=wPaper;
    MoveL Offs(pOrigin,364.33,143.12,6.00),vTravel,z5,tPen\WObj:=wPaper;
    MoveL Offs(pOrigin,364.33,143.12,0.00),v60,z0,tPen\WObj:=wPaper;
    MoveL Offs(pOrigin,364.75,143.55,0.00),v40,z0,tPen\WObj:=wPaper;
    MoveL Offs(pOrigin,364.33,143.12,0.00),v40,fine,tPen\WObj:=wPaper;
    MoveL Offs(pOrigin,364.33,143.12,6.00),v60,z5,tPen\WObj:=wPaper;
    MoveL Offs(pOrigin,363.26,141.21,6.00),vTravel,z5,tPen\WObj:=wPaper;
    MoveL Offs(pOrigin,363.26,141.21,0.00),v60,z0,tPen\WObj:=wPaper;
    MoveL Offs(pOrigin,360.92,139.73,0.00),v40,z0,tPen\WObj:=wPaper;
    MoveL Offs(pOrigin,360.08,138.45,0.00),v40,fine,tPen\WObj:=wPaper;
    MoveL Offs(pOrigin,360.08,138.45,6.00),v60,z5,tPen\WObj:=wPaper;
    MoveL Offs(pOrigin,359.01,137.39,6.00),vTravel,z5,tPen\WObj:=wPaper;
    MoveL Offs(pOrigin,359.01,137.39,0.00),v60,z0,tPen\WObj:=wPaper;
    MoveL Offs(pOrigin,359.44,137.81,0.00),v40,z0,tPen\WObj:=wPaper;
    MoveL Offs(pOrigin,359.01,137.39,0.00),v40,fine,tPen\WObj:=wPaper;
    MoveL Offs(pOrigin,359.01,137.39,6.00),v60,z5,tPen\WObj:=wPaper;
    MoveL Offs(pOrigin,357.52,129.31,6.00),vTravel,z5,tPen\WObj:=wPaper;
    MoveL Offs(pOrigin,357.52,129.31,0.00),v60,z0,tPen\WObj:=wPaper;
    MoveL Offs(pOrigin,357.95,129.74,0.00),v40,z0,tPen\WObj:=wPaper;
    MoveL Offs(pOrigin,357.52,129.31,0.00),v40,fine,tPen\WObj:=wPaper;
    MoveL Offs(pOrigin,357.52,129.31,6.00),v60,z5,tPen\WObj:=wPaper;
    MoveL Offs(pOrigin,352.85,125.06,6.00),vTravel,z5,tPen\WObj:=wPaper;
    MoveL Offs(pOrigin,352.85,125.06,0.00),v60,z0,tPen\WObj:=wPaper;
    MoveL Offs(pOrigin,353.42,125.49,0.00),v40,z0,tPen\WObj:=wPaper;
    MoveL Offs(pOrigin,356.89,130.80,0.00),v40,z0,tPen\WObj:=wPaper;
    MoveL Offs(pOrigin,361.14,135.69,0.00),v40,z0,tPen\WObj:=wPaper;
    MoveL Offs(pOrigin,366.66,140.01,0.00),v40,z0,tPen\WObj:=wPaper;
    MoveL Offs(pOrigin,370.06,141.92,0.00),v40,z0,tPen\WObj:=wPaper;
    MoveL Offs(pOrigin,371.76,142.27,0.00),v40,z0,tPen\WObj:=wPaper;
    MoveL Offs(pOrigin,371.76,142.27,0.00),v40,z0,tPen\WObj:=wPaper;
    MoveL Offs(pOrigin,377.71,144.19,0.00),v40,fine,tPen\WObj:=wPaper;
    MoveL Offs(pOrigin,377.71,144.19,6.00),v60,z5,tPen\WObj:=wPaper;
    MoveL Offs(pOrigin,379.62,141.00,6.00),vTravel,z5,tPen\WObj:=wPaper;
    MoveL Offs(pOrigin,379.62,141.00,0.00),v60,z0,tPen\WObj:=wPaper;
    MoveL Offs(pOrigin,380.05,141.21,0.00),v40,z0,tPen\WObj:=wPaper;
    MoveL Offs(pOrigin,379.62,141.00,0.00),v40,z0,tPen\WObj:=wPaper;
    MoveL Offs(pOrigin,380.26,141.43,0.00),v40,z0,tPen\WObj:=wPaper;
    MoveL Offs(pOrigin,380.90,142.06,0.00),v40,z0,tPen\WObj:=wPaper;
    MoveL Offs(pOrigin,380.26,141.43,0.00),v40,fine,tPen\WObj:=wPaper;
    MoveL Offs(pOrigin,380.26,141.43,6.00),v60,z5,tPen\WObj:=wPaper;
    MoveL Offs(pOrigin,381.96,142.91,6.00),vTravel,z5,tPen\WObj:=wPaper;
    MoveL Offs(pOrigin,381.96,142.91,0.00),v60,z0,tPen\WObj:=wPaper;
    MoveL Offs(pOrigin,384.09,144.82,0.00),v40,z0,tPen\WObj:=wPaper;
    MoveL Offs(pOrigin,381.96,142.91,0.00),v40,fine,tPen\WObj:=wPaper;
    MoveL Offs(pOrigin,381.96,142.91,6.00),v60,z5,tPen\WObj:=wPaper;
    MoveL Offs(pOrigin,384.51,145.46,6.00),vTravel,z5,tPen\WObj:=wPaper;
    MoveL Offs(pOrigin,384.51,145.46,0.00),v60,z0,tPen\WObj:=wPaper;
    MoveL Offs(pOrigin,384.94,145.89,0.00),v40,z0,tPen\WObj:=wPaper;
    MoveL Offs(pOrigin,384.51,145.46,0.00),v40,fine,tPen\WObj:=wPaper;
    MoveL Offs(pOrigin,384.51,145.46,6.00),v60,z5,tPen\WObj:=wPaper;
    MoveL Offs(pOrigin,387.49,143.34,6.00),vTravel,z5,tPen\WObj:=wPaper;
    MoveL Offs(pOrigin,387.49,143.34,0.00),v60,z0,tPen\WObj:=wPaper;
    MoveL Offs(pOrigin,387.27,143.76,0.00),v40,z0,tPen\WObj:=wPaper;
    MoveL Offs(pOrigin,387.49,143.34,0.00),v40,z0,tPen\WObj:=wPaper;
    MoveL Offs(pOrigin,388.12,142.70,0.00),v40,z0,tPen\WObj:=wPaper;
    MoveL Offs(pOrigin,387.91,143.12,0.00),v40,z0,tPen\WObj:=wPaper;
    MoveL Offs(pOrigin,388.12,142.70,0.00),v40,z0,tPen\WObj:=wPaper;
    MoveL Offs(pOrigin,388.55,142.49,0.00),v40,z0,tPen\WObj:=wPaper;
    MoveL Offs(pOrigin,388.76,142.06,0.00),v40,z0,tPen\WObj:=wPaper;
    MoveL Offs(pOrigin,388.55,142.49,0.00),v40,fine,tPen\WObj:=wPaper;
    MoveL Offs(pOrigin,388.55,142.49,6.00),v60,z5,tPen\WObj:=wPaper;
    MoveL Offs(pOrigin,389.61,141.00,6.00),vTravel,z5,tPen\WObj:=wPaper;
    MoveL Offs(pOrigin,389.61,141.00,0.00),v60,z0,tPen\WObj:=wPaper;
    MoveL Offs(pOrigin,389.40,141.43,0.00),v40,z0,tPen\WObj:=wPaper;
    MoveL Offs(pOrigin,389.61,141.00,0.00),v40,fine,tPen\WObj:=wPaper;
    MoveL Offs(pOrigin,389.61,141.00,6.00),v60,z5,tPen\WObj:=wPaper;
    MoveL Offs(pOrigin,388.27,140.15,6.00),vTravel,z5,tPen\WObj:=wPaper;
    MoveL Offs(pOrigin,388.27,140.15,0.00),v60,z0,tPen\WObj:=wPaper;
    MoveL Offs(pOrigin,385.79,142.70,0.00),v40,z0,tPen\WObj:=wPaper;
    MoveL Offs(pOrigin,388.27,140.15,0.00),v40,fine,tPen\WObj:=wPaper;
    MoveL Offs(pOrigin,388.27,140.15,6.00),v60,z5,tPen\WObj:=wPaper;
    MoveL Offs(pOrigin,387.06,137.39,6.00),vTravel,z5,tPen\WObj:=wPaper;
    MoveL Offs(pOrigin,387.06,137.39,0.00),v60,z0,tPen\WObj:=wPaper;
    MoveL Offs(pOrigin,384.09,137.39,0.00),v40,z0,tPen\WObj:=wPaper;
    MoveL Offs(pOrigin,381.11,136.54,0.00),v40,z0,tPen\WObj:=wPaper;
    MoveL Offs(pOrigin,377.08,134.70,0.00),v40,z0,tPen\WObj:=wPaper;
    MoveL Offs(pOrigin,374.95,133.35,0.00),v40,fine,tPen\WObj:=wPaper;
    MoveL Offs(pOrigin,374.95,133.35,6.00),v60,z5,tPen\WObj:=wPaper;
    MoveL Offs(pOrigin,372.61,134.20,6.00),vTravel,z5,tPen\WObj:=wPaper;
    MoveL Offs(pOrigin,372.61,134.20,0.00),v60,z0,tPen\WObj:=wPaper;
    MoveL Offs(pOrigin,375.80,137.18,0.00),v40,z0,tPen\WObj:=wPaper;
    MoveL Offs(pOrigin,377.92,138.66,0.00),v40,fine,tPen\WObj:=wPaper;
    MoveL Offs(pOrigin,377.92,138.66,6.00),v60,z5,tPen\WObj:=wPaper;
    MoveL Offs(pOrigin,375.59,136.75,6.00),vTravel,z5,tPen\WObj:=wPaper;
    MoveL Offs(pOrigin,375.59,136.75,0.00),v60,z0,tPen\WObj:=wPaper;
    MoveL Offs(pOrigin,376.01,137.18,0.00),v40,z0,tPen\WObj:=wPaper;
    MoveL Offs(pOrigin,375.59,136.75,0.00),v40,fine,tPen\WObj:=wPaper;
    MoveL Offs(pOrigin,375.59,136.75,6.00),v60,z5,tPen\WObj:=wPaper;
    MoveL Offs(pOrigin,371.76,142.27,6.00),vTravel,z5,tPen\WObj:=wPaper;
    MoveL Offs(pOrigin,371.76,142.27,0.00),v60,z0,tPen\WObj:=wPaper;
    MoveL Offs(pOrigin,371.34,141.35,0.00),v40,z0,tPen\WObj:=wPaper;
    MoveL Offs(pOrigin,369.42,140.50,0.00),v40,z0,tPen\WObj:=wPaper;
    MoveL Offs(pOrigin,364.96,137.18,0.00),v40,z0,tPen\WObj:=wPaper;
    MoveL Offs(pOrigin,360.08,132.29,0.00),v40,z0,tPen\WObj:=wPaper;
    MoveL Offs(pOrigin,357.10,128.46,0.00),v40,z0,tPen\WObj:=wPaper;
    MoveL Offs(pOrigin,354.41,124.21,0.00),v40,z0,tPen\WObj:=wPaper;
    MoveL Offs(pOrigin,351.72,118.26,0.00),v40,z0,tPen\WObj:=wPaper;
    MoveL Offs(pOrigin,350.30,112.95,0.00),v40,z0,tPen\WObj:=wPaper;
    MoveL Offs(pOrigin,350.30,111.89,0.00),v40,z0,tPen\WObj:=wPaper;
    MoveL Offs(pOrigin,350.73,111.25,0.00),v40,fine,tPen\WObj:=wPaper;
    MoveL Offs(pOrigin,350.73,111.25,6.00),v60,z5,tPen\WObj:=wPaper;
    MoveL Offs(pOrigin,353.49,109.55,6.00),vTravel,z5,tPen\WObj:=wPaper;
    MoveL Offs(pOrigin,353.49,109.55,0.00),v60,z0,tPen\WObj:=wPaper;
    MoveL Offs(pOrigin,354.34,110.40,0.00),v40,z0,tPen\WObj:=wPaper;
    MoveL Offs(pOrigin,353.49,109.55,0.00),v40,fine,tPen\WObj:=wPaper;
    MoveL Offs(pOrigin,353.49,109.55,6.00),v60,z5,tPen\WObj:=wPaper;
    MoveL Offs(pOrigin,354.76,110.61,6.00),vTravel,z5,tPen\WObj:=wPaper;
  ENDPROC

  PROC DrawPart88()
    MoveL Offs(pOrigin,354.76,110.61,0.00),v60,z0,tPen\WObj:=wPaper;
    MoveL Offs(pOrigin,355.40,111.25,0.00),v40,z0,tPen\WObj:=wPaper;
    MoveL Offs(pOrigin,354.76,110.61,0.00),v40,fine,tPen\WObj:=wPaper;
    MoveL Offs(pOrigin,354.76,110.61,6.00),v60,z5,tPen\WObj:=wPaper;
    MoveL Offs(pOrigin,356.67,108.28,6.00),vTravel,z5,tPen\WObj:=wPaper;
    MoveL Offs(pOrigin,356.67,108.28,0.00),v60,z0,tPen\WObj:=wPaper;
    MoveL Offs(pOrigin,357.52,109.12,0.00),v40,z0,tPen\WObj:=wPaper;
    MoveL Offs(pOrigin,358.59,109.34,0.00),v40,fine,tPen\WObj:=wPaper;
    MoveL Offs(pOrigin,358.59,109.34,6.00),v60,z5,tPen\WObj:=wPaper;
    MoveL Offs(pOrigin,356.67,108.28,6.00),vTravel,z5,tPen\WObj:=wPaper;
    MoveL Offs(pOrigin,356.67,108.28,0.00),v60,z0,tPen\WObj:=wPaper;
    MoveL Offs(pOrigin,352.64,105.30,0.00),v40,z0,tPen\WObj:=wPaper;
    MoveL Offs(pOrigin,350.51,103.18,0.00),v40,z0,tPen\WObj:=wPaper;
    MoveL Offs(pOrigin,349.52,102.96,0.00),v40,z0,tPen\WObj:=wPaper;
    MoveL Offs(pOrigin,349.45,104.03,0.00),v40,z0,tPen\WObj:=wPaper;
    MoveL Offs(pOrigin,350.02,105.72,0.00),v40,z0,tPen\WObj:=wPaper;
    MoveL Offs(pOrigin,351.15,107.43,0.00),v40,z0,tPen\WObj:=wPaper;
    MoveL Offs(pOrigin,354.12,110.40,0.00),v40,z0,tPen\WObj:=wPaper;
    MoveL Offs(pOrigin,358.38,113.45,0.00),v40,z0,tPen\WObj:=wPaper;
    MoveL Offs(pOrigin,358.59,114.01,0.00),v40,z0,tPen\WObj:=wPaper;
    MoveL Offs(pOrigin,358.59,114.01,0.00),v40,z0,tPen\WObj:=wPaper;
    MoveL Offs(pOrigin,359.44,114.01,0.00),v40,z0,tPen\WObj:=wPaper;
    MoveL Offs(pOrigin,359.86,114.86,0.00),v40,z0,tPen\WObj:=wPaper;
    MoveL Offs(pOrigin,359.86,114.86,0.00),v40,z0,tPen\WObj:=wPaper;
    MoveL Offs(pOrigin,365.39,117.34,0.00),v40,z0,tPen\WObj:=wPaper;
    MoveL Offs(pOrigin,369.21,118.62,0.00),v40,z0,tPen\WObj:=wPaper;
    MoveL Offs(pOrigin,369.64,118.47,0.00),v40,fine,tPen\WObj:=wPaper;
    MoveL Offs(pOrigin,369.64,118.47,6.00),v60,z5,tPen\WObj:=wPaper;
    MoveL Offs(pOrigin,362.41,124.85,6.00),vTravel,z5,tPen\WObj:=wPaper;
    MoveL Offs(pOrigin,362.41,124.85,0.00),v60,z0,tPen\WObj:=wPaper;
    MoveL Offs(pOrigin,363.26,125.49,0.00),v40,z0,tPen\WObj:=wPaper;
    MoveL Offs(pOrigin,362.41,124.85,0.00),v40,fine,tPen\WObj:=wPaper;
    MoveL Offs(pOrigin,362.41,124.85,6.00),v60,z5,tPen\WObj:=wPaper;
    MoveL Offs(pOrigin,368.79,128.89,6.00),vTravel,z5,tPen\WObj:=wPaper;
    MoveL Offs(pOrigin,368.79,128.89,0.00),v60,z0,tPen\WObj:=wPaper;
    MoveL Offs(pOrigin,364.33,126.12,0.00),v40,z0,tPen\WObj:=wPaper;
    MoveL Offs(pOrigin,361.56,124.00,0.00),v40,z0,tPen\WObj:=wPaper;
    MoveL Offs(pOrigin,357.74,120.39,0.00),v40,z0,tPen\WObj:=wPaper;
    MoveL Offs(pOrigin,355.40,117.41,0.00),v40,z0,tPen\WObj:=wPaper;
    MoveL Offs(pOrigin,355.40,117.41,0.00),v40,z0,tPen\WObj:=wPaper;
    MoveL Offs(pOrigin,354.34,117.20,0.00),v40,z0,tPen\WObj:=wPaper;
    MoveL Offs(pOrigin,354.12,116.56,0.00),v40,z0,tPen\WObj:=wPaper;
    MoveL Offs(pOrigin,354.12,116.56,0.00),v40,z0,tPen\WObj:=wPaper;
    MoveL Offs(pOrigin,353.70,116.35,0.00),v40,z0,tPen\WObj:=wPaper;
    MoveL Offs(pOrigin,353.49,115.29,0.00),v40,z0,tPen\WObj:=wPaper;
    MoveL Offs(pOrigin,353.49,115.29,0.00),v40,z0,tPen\WObj:=wPaper;
    MoveL Offs(pOrigin,354.34,115.50,0.00),v40,z0,tPen\WObj:=wPaper;
    MoveL Offs(pOrigin,354.55,116.35,0.00),v40,z0,tPen\WObj:=wPaper;
    MoveL Offs(pOrigin,354.55,116.35,0.00),v40,z0,tPen\WObj:=wPaper;
    MoveL Offs(pOrigin,355.19,116.35,0.00),v40,z0,tPen\WObj:=wPaper;
    MoveL Offs(pOrigin,355.40,117.41,0.00),v40,fine,tPen\WObj:=wPaper;
    MoveL Offs(pOrigin,355.40,117.41,6.00),v60,z5,tPen\WObj:=wPaper;
    MoveL Offs(pOrigin,356.89,119.54,6.00),vTravel,z5,tPen\WObj:=wPaper;
    MoveL Offs(pOrigin,356.89,119.54,0.00),v60,z0,tPen\WObj:=wPaper;
    MoveL Offs(pOrigin,357.31,119.96,0.00),v40,z0,tPen\WObj:=wPaper;
    MoveL Offs(pOrigin,356.89,119.54,0.00),v40,fine,tPen\WObj:=wPaper;
    MoveL Offs(pOrigin,356.89,119.54,6.00),v60,z5,tPen\WObj:=wPaper;
    MoveL Offs(pOrigin,358.59,114.44,6.00),vTravel,z5,tPen\WObj:=wPaper;
    MoveL Offs(pOrigin,358.59,114.44,0.00),v60,z0,tPen\WObj:=wPaper;
    MoveL Offs(pOrigin,356.46,113.45,0.00),v40,z0,tPen\WObj:=wPaper;
    MoveL Offs(pOrigin,352.42,110.54,0.00),v40,z0,tPen\WObj:=wPaper;
    MoveL Offs(pOrigin,351.15,110.26,0.00),v40,z0,tPen\WObj:=wPaper;
    MoveL Offs(pOrigin,350.80,111.04,0.00),v40,z0,tPen\WObj:=wPaper;
    MoveL Offs(pOrigin,353.49,115.29,0.00),v40,z0,tPen\WObj:=wPaper;
    MoveL Offs(pOrigin,353.27,114.86,0.00),v40,z0,tPen\WObj:=wPaper;
    MoveL Offs(pOrigin,353.49,115.29,0.00),v40,z0,tPen\WObj:=wPaper;
    MoveL Offs(pOrigin,353.27,114.86,0.00),v40,z0,tPen\WObj:=wPaper;
    MoveL Offs(pOrigin,352.85,114.22,0.00),v40,z0,tPen\WObj:=wPaper;
    MoveL Offs(pOrigin,353.06,114.65,0.00),v40,z0,tPen\WObj:=wPaper;
    MoveL Offs(pOrigin,352.85,114.22,0.00),v40,fine,tPen\WObj:=wPaper;
    MoveL Offs(pOrigin,352.85,114.22,6.00),v60,z5,tPen\WObj:=wPaper;
    MoveL Offs(pOrigin,358.59,114.44,6.00),vTravel,z5,tPen\WObj:=wPaper;
    MoveL Offs(pOrigin,358.59,114.44,0.00),v60,z0,tPen\WObj:=wPaper;
    MoveL Offs(pOrigin,358.80,114.86,0.00),v40,z0,tPen\WObj:=wPaper;
    MoveL Offs(pOrigin,359.44,115.07,0.00),v40,z0,tPen\WObj:=wPaper;
    MoveL Offs(pOrigin,359.86,114.86,0.00),v40,fine,tPen\WObj:=wPaper;
    MoveL Offs(pOrigin,359.86,114.86,6.00),v60,z5,tPen\WObj:=wPaper;
    MoveL Offs(pOrigin,354.76,107.21,6.00),vTravel,z5,tPen\WObj:=wPaper;
    MoveL Offs(pOrigin,354.76,107.21,0.00),v60,z0,tPen\WObj:=wPaper;
    MoveL Offs(pOrigin,355.40,107.64,0.00),v40,z0,tPen\WObj:=wPaper;
    MoveL Offs(pOrigin,354.76,107.21,0.00),v40,fine,tPen\WObj:=wPaper;
    MoveL Offs(pOrigin,354.76,107.21,6.00),v60,z5,tPen\WObj:=wPaper;
    MoveL Offs(pOrigin,354.76,105.72,6.00),vTravel,z5,tPen\WObj:=wPaper;
    MoveL Offs(pOrigin,354.76,105.72,0.00),v60,z0,tPen\WObj:=wPaper;
    MoveL Offs(pOrigin,355.40,106.36,0.00),v40,z0,tPen\WObj:=wPaper;
    MoveL Offs(pOrigin,354.76,105.72,0.00),v40,fine,tPen\WObj:=wPaper;
    MoveL Offs(pOrigin,354.76,105.72,6.00),v60,z5,tPen\WObj:=wPaper;
    MoveL Offs(pOrigin,353.49,104.66,6.00),vTravel,z5,tPen\WObj:=wPaper;
    MoveL Offs(pOrigin,353.49,104.66,0.00),v60,z0,tPen\WObj:=wPaper;
    MoveL Offs(pOrigin,354.34,105.51,0.00),v40,z0,tPen\WObj:=wPaper;
    MoveL Offs(pOrigin,353.49,104.66,0.00),v40,z0,tPen\WObj:=wPaper;
    MoveL Offs(pOrigin,353.06,105.72,0.00),v40,z0,tPen\WObj:=wPaper;
    MoveL Offs(pOrigin,353.70,106.36,0.00),v40,z0,tPen\WObj:=wPaper;
    MoveL Offs(pOrigin,353.06,105.72,0.00),v40,fine,tPen\WObj:=wPaper;
    MoveL Offs(pOrigin,353.06,105.72,6.00),v60,z5,tPen\WObj:=wPaper;
    MoveL Offs(pOrigin,351.79,104.66,6.00),vTravel,z5,tPen\WObj:=wPaper;
    MoveL Offs(pOrigin,351.79,104.66,0.00),v60,z0,tPen\WObj:=wPaper;
    MoveL Offs(pOrigin,352.64,105.51,0.00),v40,z0,tPen\WObj:=wPaper;
    MoveL Offs(pOrigin,351.79,104.66,0.00),v40,fine,tPen\WObj:=wPaper;
    MoveL Offs(pOrigin,351.79,104.66,6.00),v60,z5,tPen\WObj:=wPaper;
    MoveL Offs(pOrigin,352.00,103.18,6.00),vTravel,z5,tPen\WObj:=wPaper;
    MoveL Offs(pOrigin,352.00,103.18,0.00),v60,z0,tPen\WObj:=wPaper;
    MoveL Offs(pOrigin,352.85,104.03,0.00),v40,z0,tPen\WObj:=wPaper;
    MoveL Offs(pOrigin,352.00,103.18,0.00),v40,fine,tPen\WObj:=wPaper;
    MoveL Offs(pOrigin,352.00,103.18,6.00),v60,z5,tPen\WObj:=wPaper;
    MoveL Offs(pOrigin,350.30,103.18,6.00),vTravel,z5,tPen\WObj:=wPaper;
    MoveL Offs(pOrigin,350.30,103.18,0.00),v60,z0,tPen\WObj:=wPaper;
    MoveL Offs(pOrigin,351.15,104.03,0.00),v40,z0,tPen\WObj:=wPaper;
    MoveL Offs(pOrigin,350.30,103.18,0.00),v40,fine,tPen\WObj:=wPaper;
    MoveL Offs(pOrigin,350.30,103.18,6.00),v60,z5,tPen\WObj:=wPaper;
    MoveL Offs(pOrigin,350.51,101.69,6.00),vTravel,z5,tPen\WObj:=wPaper;
    MoveL Offs(pOrigin,350.51,101.69,0.00),v60,z0,tPen\WObj:=wPaper;
    MoveL Offs(pOrigin,351.36,102.54,0.00),v40,z0,tPen\WObj:=wPaper;
    MoveL Offs(pOrigin,350.51,101.69,0.00),v40,fine,tPen\WObj:=wPaper;
    MoveL Offs(pOrigin,350.51,101.69,6.00),v60,z5,tPen\WObj:=wPaper;
    MoveL Offs(pOrigin,349.66,100.41,6.00),vTravel,z5,tPen\WObj:=wPaper;
    MoveL Offs(pOrigin,349.66,100.41,0.00),v60,z0,tPen\WObj:=wPaper;
    MoveL Offs(pOrigin,350.30,101.26,0.00),v40,z0,tPen\WObj:=wPaper;
    MoveL Offs(pOrigin,349.66,100.41,0.00),v40,fine,tPen\WObj:=wPaper;
    MoveL Offs(pOrigin,349.66,100.41,6.00),v60,z5,tPen\WObj:=wPaper;
  ENDPROC

  PROC DrawPart89()
    MoveL Offs(pOrigin,347.54,105.72,6.00),vTravel,z5,tPen\WObj:=wPaper;
    MoveL Offs(pOrigin,347.54,105.72,0.00),v60,z0,tPen\WObj:=wPaper;
    MoveL Offs(pOrigin,346.33,101.47,0.00),v40,z0,tPen\WObj:=wPaper;
    MoveL Offs(pOrigin,345.55,100.41,0.00),v40,z0,tPen\WObj:=wPaper;
    MoveL Offs(pOrigin,342.79,93.40,0.00),v40,z0,tPen\WObj:=wPaper;
    MoveL Offs(pOrigin,342.23,93.12,0.00),v40,z0,tPen\WObj:=wPaper;
    MoveL Offs(pOrigin,342.01,93.61,0.00),v40,z0,tPen\WObj:=wPaper;
    MoveL Offs(pOrigin,344.42,99.99,0.00),v40,z0,tPen\WObj:=wPaper;
    MoveL Offs(pOrigin,348.17,111.68,0.00),v40,z0,tPen\WObj:=wPaper;
    MoveL Offs(pOrigin,353.91,139.30,0.00),v40,z0,tPen\WObj:=wPaper;
    MoveL Offs(pOrigin,360.50,165.23,0.00),v40,z0,tPen\WObj:=wPaper;
    MoveL Offs(pOrigin,365.53,181.16,0.00),v40,z0,tPen\WObj:=wPaper;
    MoveL Offs(pOrigin,366.95,184.56,0.00),v40,z0,tPen\WObj:=wPaper;
    MoveL Offs(pOrigin,369.85,189.45,0.00),v40,z0,tPen\WObj:=wPaper;
    MoveL Offs(pOrigin,369.64,189.80,0.00),v40,z0,tPen\WObj:=wPaper;
    MoveL Offs(pOrigin,365.60,191.15,0.00),v40,z0,tPen\WObj:=wPaper;
    MoveL Offs(pOrigin,342.86,197.31,0.00),v40,z0,tPen\WObj:=wPaper;
    MoveL Offs(pOrigin,333.94,200.43,0.00),v40,z0,tPen\WObj:=wPaper;
    MoveL Offs(pOrigin,317.58,207.37,0.00),v40,z0,tPen\WObj:=wPaper;
    MoveL Offs(pOrigin,309.50,210.06,0.00),v40,z0,tPen\WObj:=wPaper;
    MoveL Offs(pOrigin,303.41,211.48,0.00),v40,z0,tPen\WObj:=wPaper;
    MoveL Offs(pOrigin,303.83,210.27,0.00),v40,z0,tPen\WObj:=wPaper;
    MoveL Offs(pOrigin,308.01,205.25,0.00),v40,z0,tPen\WObj:=wPaper;
    MoveL Offs(pOrigin,312.69,204.54,0.00),v40,z0,tPen\WObj:=wPaper;
    MoveL Offs(pOrigin,317.79,203.26,0.00),v40,z0,tPen\WObj:=wPaper;
    MoveL Offs(pOrigin,321.83,201.92,0.00),v40,z0,tPen\WObj:=wPaper;
    MoveL Offs(pOrigin,322.25,201.35,0.00),v40,z0,tPen\WObj:=wPaper;
    MoveL Offs(pOrigin,322.25,201.35,0.00),v40,z0,tPen\WObj:=wPaper;
    MoveL Offs(pOrigin,336.27,196.46,0.00),v40,z0,tPen\WObj:=wPaper;
    MoveL Offs(pOrigin,337.34,196.46,0.00),v40,fine,tPen\WObj:=wPaper;
    MoveL Offs(pOrigin,337.34,196.46,6.00),v60,z5,tPen\WObj:=wPaper;
    MoveL Offs(pOrigin,327.77,204.75,6.00),vTravel,z5,tPen\WObj:=wPaper;
    MoveL Offs(pOrigin,327.77,204.75,0.00),v60,z0,tPen\WObj:=wPaper;
    MoveL Offs(pOrigin,328.20,204.54,0.00),v40,z0,tPen\WObj:=wPaper;
    MoveL Offs(pOrigin,327.77,204.75,0.00),v40,fine,tPen\WObj:=wPaper;
    MoveL Offs(pOrigin,327.77,204.75,6.00),v60,z5,tPen\WObj:=wPaper;
    MoveL Offs(pOrigin,323.31,206.66,6.00),vTravel,z5,tPen\WObj:=wPaper;
    MoveL Offs(pOrigin,323.31,206.66,0.00),v60,z0,tPen\WObj:=wPaper;
    MoveL Offs(pOrigin,323.74,206.45,0.00),v40,z0,tPen\WObj:=wPaper;
    MoveL Offs(pOrigin,323.31,206.66,0.00),v40,fine,tPen\WObj:=wPaper;
    MoveL Offs(pOrigin,323.31,206.66,6.00),v60,z5,tPen\WObj:=wPaper;
    MoveL Offs(pOrigin,322.25,201.35,6.00),vTravel,z5,tPen\WObj:=wPaper;
    MoveL Offs(pOrigin,322.25,201.35,0.00),v60,z0,tPen\WObj:=wPaper;
    MoveL Offs(pOrigin,321.61,201.14,0.00),v40,z0,tPen\WObj:=wPaper;
    MoveL Offs(pOrigin,313.96,203.26,0.00),v40,z0,tPen\WObj:=wPaper;
    MoveL Offs(pOrigin,309.92,204.11,0.00),v40,z0,tPen\WObj:=wPaper;
    MoveL Offs(pOrigin,309.36,203.90,0.00),v40,z0,tPen\WObj:=wPaper;
    MoveL Offs(pOrigin,313.18,198.59,0.00),v40,z0,tPen\WObj:=wPaper;
    MoveL Offs(pOrigin,316.80,194.55,0.00),v40,z0,tPen\WObj:=wPaper;
    MoveL Offs(pOrigin,318.71,191.57,0.00),v40,z0,tPen\WObj:=wPaper;
    MoveL Offs(pOrigin,320.41,186.05,0.00),v40,z0,tPen\WObj:=wPaper;
    MoveL Offs(pOrigin,320.98,185.20,0.00),v40,z0,tPen\WObj:=wPaper;
    MoveL Offs(pOrigin,320.55,184.56,0.00),v40,z0,tPen\WObj:=wPaper;
    MoveL Offs(pOrigin,320.55,184.56,0.00),v40,z0,tPen\WObj:=wPaper;
    MoveL Offs(pOrigin,320.55,183.50,0.00),v40,z0,tPen\WObj:=wPaper;
    MoveL Offs(pOrigin,320.55,183.50,0.00),v40,z0,tPen\WObj:=wPaper;
    MoveL Offs(pOrigin,321.19,182.86,0.00),v40,z0,tPen\WObj:=wPaper;
    MoveL Offs(pOrigin,320.55,181.59,0.00),v40,z0,tPen\WObj:=wPaper;
    MoveL Offs(pOrigin,320.55,179.25,0.00),v40,z0,tPen\WObj:=wPaper;
    MoveL Offs(pOrigin,318.00,170.32,0.00),v40,fine,tPen\WObj:=wPaper;
    MoveL Offs(pOrigin,318.00,170.32,6.00),v60,z5,tPen\WObj:=wPaper;
    MoveL Offs(pOrigin,320.55,182.01,6.00),vTravel,z5,tPen\WObj:=wPaper;
    MoveL Offs(pOrigin,320.55,182.01,0.00),v60,z0,tPen\WObj:=wPaper;
    MoveL Offs(pOrigin,320.34,183.29,0.00),v40,z0,tPen\WObj:=wPaper;
    MoveL Offs(pOrigin,320.55,183.50,0.00),v40,z0,tPen\WObj:=wPaper;
    MoveL Offs(pOrigin,320.55,184.56,0.00),v40,z0,tPen\WObj:=wPaper;
    MoveL Offs(pOrigin,320.12,184.99,0.00),v40,z0,tPen\WObj:=wPaper;
    MoveL Offs(pOrigin,320.34,185.84,0.00),v40,fine,tPen\WObj:=wPaper;
    MoveL Offs(pOrigin,320.34,185.84,6.00),v60,z5,tPen\WObj:=wPaper;
    MoveL Offs(pOrigin,318.64,191.36,6.00),vTravel,z5,tPen\WObj:=wPaper;
    MoveL Offs(pOrigin,318.64,191.36,0.00),v60,z0,tPen\WObj:=wPaper;
    MoveL Offs(pOrigin,318.42,191.79,0.00),v40,z0,tPen\WObj:=wPaper;
    MoveL Offs(pOrigin,318.64,191.36,0.00),v40,fine,tPen\WObj:=wPaper;
    MoveL Offs(pOrigin,318.64,191.36,6.00),v60,z5,tPen\WObj:=wPaper;
    MoveL Offs(pOrigin,318.00,192.43,6.00),vTravel,z5,tPen\WObj:=wPaper;
    MoveL Offs(pOrigin,318.00,192.43,0.00),v60,z0,tPen\WObj:=wPaper;
    MoveL Offs(pOrigin,317.79,192.85,0.00),v40,z0,tPen\WObj:=wPaper;
    MoveL Offs(pOrigin,318.00,192.43,0.00),v40,fine,tPen\WObj:=wPaper;
    MoveL Offs(pOrigin,318.00,192.43,6.00),v60,z5,tPen\WObj:=wPaper;
    MoveL Offs(pOrigin,316.09,194.98,6.00),vTravel,z5,tPen\WObj:=wPaper;
    MoveL Offs(pOrigin,316.09,194.98,0.00),v60,z0,tPen\WObj:=wPaper;
    MoveL Offs(pOrigin,314.39,193.56,0.00),v40,z0,tPen\WObj:=wPaper;
    MoveL Offs(pOrigin,306.95,190.16,0.00),v40,z0,tPen\WObj:=wPaper;
    MoveL Offs(pOrigin,303.90,188.39,0.00),v40,z0,tPen\WObj:=wPaper;
    MoveL Offs(pOrigin,304.40,187.89,0.00),v40,z0,tPen\WObj:=wPaper;
    MoveL Offs(pOrigin,318.21,183.15,0.00),v40,z0,tPen\WObj:=wPaper;
    MoveL Offs(pOrigin,318.64,182.65,0.00),v40,z0,tPen\WObj:=wPaper;
    MoveL Offs(pOrigin,318.64,181.59,0.00),v40,z0,tPen\WObj:=wPaper;
    MoveL Offs(pOrigin,310.35,156.51,0.00),v40,z0,tPen\WObj:=wPaper;
    MoveL Offs(pOrigin,298.38,117.62,0.00),v40,z0,tPen\WObj:=wPaper;
    MoveL Offs(pOrigin,298.66,117.41,0.00),v40,z0,tPen\WObj:=wPaper;
    MoveL Offs(pOrigin,322.04,123.79,0.00),v40,z0,tPen\WObj:=wPaper;
    MoveL Offs(pOrigin,331.60,126.55,0.00),v40,z0,tPen\WObj:=wPaper;
    MoveL Offs(pOrigin,335.00,128.04,0.00),v40,z0,tPen\WObj:=wPaper;
    MoveL Offs(pOrigin,335.00,128.04,0.00),v40,z0,tPen\WObj:=wPaper;
    MoveL Offs(pOrigin,336.06,127.82,0.00),v40,z0,tPen\WObj:=wPaper;
    MoveL Offs(pOrigin,344.56,130.38,0.00),v40,z0,tPen\WObj:=wPaper;
    MoveL Offs(pOrigin,345.20,130.09,0.00),v40,z0,tPen\WObj:=wPaper;
    MoveL Offs(pOrigin,345.62,128.46,0.00),v40,z0,tPen\WObj:=wPaper;
    MoveL Offs(pOrigin,345.84,124.85,0.00),v40,z0,tPen\WObj:=wPaper;
    MoveL Offs(pOrigin,345.62,119.32,0.00),v40,z0,tPen\WObj:=wPaper;
    MoveL Offs(pOrigin,345.34,118.69,0.00),v40,z0,tPen\WObj:=wPaper;
    MoveL Offs(pOrigin,344.35,117.98,0.00),v40,z0,tPen\WObj:=wPaper;
    MoveL Offs(pOrigin,339.46,116.35,0.00),v40,z0,tPen\WObj:=wPaper;
    MoveL Offs(pOrigin,318.21,110.40,0.00),v40,z0,tPen\WObj:=wPaper;
    MoveL Offs(pOrigin,297.60,105.51,0.00),v40,z0,tPen\WObj:=wPaper;
    MoveL Offs(pOrigin,297.17,106.15,0.00),v40,z0,tPen\WObj:=wPaper;
    MoveL Offs(pOrigin,297.17,106.15,0.00),v40,z0,tPen\WObj:=wPaper;
    MoveL Offs(pOrigin,324.38,112.95,0.00),v40,z0,tPen\WObj:=wPaper;
    MoveL Offs(pOrigin,343.71,118.62,0.00),v40,z0,tPen\WObj:=wPaper;
    MoveL Offs(pOrigin,344.49,119.11,0.00),v40,z0,tPen\WObj:=wPaper;
    MoveL Offs(pOrigin,344.77,119.75,0.00),v40,z0,tPen\WObj:=wPaper;
    MoveL Offs(pOrigin,344.56,128.89,0.00),v40,z0,tPen\WObj:=wPaper;
    MoveL Offs(pOrigin,344.35,129.10,0.00),v40,z0,tPen\WObj:=wPaper;
    MoveL Offs(pOrigin,342.86,128.89,0.00),v40,z0,tPen\WObj:=wPaper;
    MoveL Offs(pOrigin,298.02,116.07,0.00),v40,z0,tPen\WObj:=wPaper;
    MoveL Offs(pOrigin,297.53,115.50,0.00),v40,z0,tPen\WObj:=wPaper;
    MoveL Offs(pOrigin,295.05,107.43,0.00),v40,z0,tPen\WObj:=wPaper;
    MoveL Offs(pOrigin,295.26,106.15,0.00),v40,z0,tPen\WObj:=wPaper;
    MoveL Offs(pOrigin,296.11,105.94,0.00),v40,z0,tPen\WObj:=wPaper;
  ENDPROC

  PROC DrawPart90()
    MoveL Offs(pOrigin,296.11,105.94,0.00),v40,z0,tPen\WObj:=wPaper;
    MoveL Offs(pOrigin,297.17,106.15,0.00),v40,z0,tPen\WObj:=wPaper;
    MoveL Offs(pOrigin,297.17,105.51,0.00),v40,z0,tPen\WObj:=wPaper;
    MoveL Offs(pOrigin,296.11,105.30,0.00),v40,fine,tPen\WObj:=wPaper;
    MoveL Offs(pOrigin,296.11,105.30,6.00),v60,z5,tPen\WObj:=wPaper;
    MoveL Offs(pOrigin,300.15,114.86,6.00),vTravel,z5,tPen\WObj:=wPaper;
    MoveL Offs(pOrigin,300.15,114.86,0.00),v60,z0,tPen\WObj:=wPaper;
    MoveL Offs(pOrigin,333.73,123.79,0.00),v40,z0,tPen\WObj:=wPaper;
    MoveL Offs(pOrigin,342.23,126.34,0.00),v40,fine,tPen\WObj:=wPaper;
    MoveL Offs(pOrigin,342.23,126.34,6.00),v60,z5,tPen\WObj:=wPaper;
    MoveL Offs(pOrigin,344.99,130.38,6.00),vTravel,z5,tPen\WObj:=wPaper;
    MoveL Offs(pOrigin,344.99,130.38,0.00),v60,z0,tPen\WObj:=wPaper;
    MoveL Offs(pOrigin,345.20,129.95,0.00),v40,z0,tPen\WObj:=wPaper;
    MoveL Offs(pOrigin,344.99,130.38,0.00),v40,fine,tPen\WObj:=wPaper;
    MoveL Offs(pOrigin,344.99,130.38,6.00),v60,z5,tPen\WObj:=wPaper;
    MoveL Offs(pOrigin,342.23,134.62,6.00),vTravel,z5,tPen\WObj:=wPaper;
    MoveL Offs(pOrigin,342.23,134.62,0.00),v60,z0,tPen\WObj:=wPaper;
    MoveL Offs(pOrigin,342.65,134.84,0.00),v40,z0,tPen\WObj:=wPaper;
    MoveL Offs(pOrigin,342.23,134.62,0.00),v40,fine,tPen\WObj:=wPaper;
    MoveL Offs(pOrigin,342.23,134.62,6.00),v60,z5,tPen\WObj:=wPaper;
    MoveL Offs(pOrigin,336.70,130.16,6.00),vTravel,z5,tPen\WObj:=wPaper;
    MoveL Offs(pOrigin,336.70,130.16,0.00),v60,z0,tPen\WObj:=wPaper;
    MoveL Offs(pOrigin,337.12,130.59,0.00),v40,z0,tPen\WObj:=wPaper;
    MoveL Offs(pOrigin,336.70,130.16,0.00),v40,fine,tPen\WObj:=wPaper;
    MoveL Offs(pOrigin,336.70,130.16,6.00),v60,z5,tPen\WObj:=wPaper;
    MoveL Offs(pOrigin,335.00,128.04,6.00),vTravel,z5,tPen\WObj:=wPaper;
    MoveL Offs(pOrigin,335.00,128.04,0.00),v60,z0,tPen\WObj:=wPaper;
    MoveL Offs(pOrigin,335.21,128.68,0.00),v40,z0,tPen\WObj:=wPaper;
    MoveL Offs(pOrigin,339.89,132.71,0.00),v40,z0,tPen\WObj:=wPaper;
    MoveL Offs(pOrigin,348.39,138.45,0.00),v40,fine,tPen\WObj:=wPaper;
    MoveL Offs(pOrigin,348.39,138.45,6.00),v60,z5,tPen\WObj:=wPaper;
    MoveL Offs(pOrigin,351.79,107.85,6.00),vTravel,z5,tPen\WObj:=wPaper;
    MoveL Offs(pOrigin,351.79,107.85,0.00),v60,z0,tPen\WObj:=wPaper;
    MoveL Offs(pOrigin,353.27,109.34,0.00),v40,z0,tPen\WObj:=wPaper;
    MoveL Offs(pOrigin,351.79,107.85,0.00),v40,z0,tPen\WObj:=wPaper;
    MoveL Offs(pOrigin,351.15,107.21,0.00),v40,z0,tPen\WObj:=wPaper;
    MoveL Offs(pOrigin,351.58,107.64,0.00),v40,z0,tPen\WObj:=wPaper;
    MoveL Offs(pOrigin,351.15,107.21,0.00),v40,fine,tPen\WObj:=wPaper;
    MoveL Offs(pOrigin,351.15,107.21,6.00),v60,z5,tPen\WObj:=wPaper;
    MoveL Offs(pOrigin,361.77,100.41,6.00),vTravel,z5,tPen\WObj:=wPaper;
    MoveL Offs(pOrigin,361.77,100.41,0.00),v60,z0,tPen\WObj:=wPaper;
    MoveL Offs(pOrigin,362.20,100.84,0.00),v40,z0,tPen\WObj:=wPaper;
    MoveL Offs(pOrigin,361.77,100.41,0.00),v40,fine,tPen\WObj:=wPaper;
    MoveL Offs(pOrigin,361.77,100.41,6.00),v60,z5,tPen\WObj:=wPaper;
    MoveL Offs(pOrigin,365.39,102.75,6.00),vTravel,z5,tPen\WObj:=wPaper;
    MoveL Offs(pOrigin,365.39,102.75,0.00),v60,z0,tPen\WObj:=wPaper;
    MoveL Offs(pOrigin,363.69,101.90,0.00),v40,z0,tPen\WObj:=wPaper;
    MoveL Offs(pOrigin,361.56,99.99,0.00),v40,z0,tPen\WObj:=wPaper;
    MoveL Offs(pOrigin,359.37,96.80,0.00),v40,z0,tPen\WObj:=wPaper;
    MoveL Offs(pOrigin,358.80,95.31,0.00),v40,fine,tPen\WObj:=wPaper;
    MoveL Offs(pOrigin,358.80,95.31,6.00),v60,z5,tPen\WObj:=wPaper;
    MoveL Offs(pOrigin,360.08,88.94,6.00),vTravel,z5,tPen\WObj:=wPaper;
    MoveL Offs(pOrigin,360.08,88.94,0.00),v60,z0,tPen\WObj:=wPaper;
    MoveL Offs(pOrigin,361.35,90.21,0.00),v40,z0,tPen\WObj:=wPaper;
    MoveL Offs(pOrigin,360.08,88.94,0.00),v40,fine,tPen\WObj:=wPaper;
    MoveL Offs(pOrigin,360.08,88.94,6.00),v60,z5,tPen\WObj:=wPaper;
    MoveL Offs(pOrigin,357.10,84.90,6.00),vTravel,z5,tPen\WObj:=wPaper;
    MoveL Offs(pOrigin,357.10,84.90,0.00),v60,z0,tPen\WObj:=wPaper;
    MoveL Offs(pOrigin,360.08,89.15,0.00),v40,z0,tPen\WObj:=wPaper;
    MoveL Offs(pOrigin,364.75,93.40,0.00),v40,z0,tPen\WObj:=wPaper;
    MoveL Offs(pOrigin,369.21,95.88,0.00),v40,z0,tPen\WObj:=wPaper;
    MoveL Offs(pOrigin,376.01,97.86,0.00),v40,fine,tPen\WObj:=wPaper;
    MoveL Offs(pOrigin,376.01,97.86,6.00),v60,z5,tPen\WObj:=wPaper;
    MoveL Offs(pOrigin,368.79,91.28,6.00),vTravel,z5,tPen\WObj:=wPaper;
    MoveL Offs(pOrigin,368.79,91.28,0.00),v60,z0,tPen\WObj:=wPaper;
    MoveL Offs(pOrigin,367.94,91.13,0.00),v40,z0,tPen\WObj:=wPaper;
    MoveL Offs(pOrigin,365.81,89.79,0.00),v40,z0,tPen\WObj:=wPaper;
    MoveL Offs(pOrigin,361.99,86.60,0.00),v40,z0,tPen\WObj:=wPaper;
    MoveL Offs(pOrigin,358.80,83.20,0.00),v40,z0,tPen\WObj:=wPaper;
    MoveL Offs(pOrigin,355.40,77.89,0.00),v40,fine,tPen\WObj:=wPaper;
    MoveL Offs(pOrigin,355.40,77.89,6.00),v60,z5,tPen\WObj:=wPaper;
    MoveL Offs(pOrigin,356.46,80.01,6.00),vTravel,z5,tPen\WObj:=wPaper;
    MoveL Offs(pOrigin,356.46,80.01,0.00),v60,z0,tPen\WObj:=wPaper;
    MoveL Offs(pOrigin,356.67,80.44,0.00),v40,z0,tPen\WObj:=wPaper;
    MoveL Offs(pOrigin,356.46,80.01,0.00),v40,fine,tPen\WObj:=wPaper;
    MoveL Offs(pOrigin,356.46,80.01,6.00),v60,z5,tPen\WObj:=wPaper;
    MoveL Offs(pOrigin,367.73,80.01,6.00),vTravel,z5,tPen\WObj:=wPaper;
    MoveL Offs(pOrigin,367.73,80.01,0.00),v60,z0,tPen\WObj:=wPaper;
    MoveL Offs(pOrigin,371.76,80.44,0.00),v40,z0,tPen\WObj:=wPaper;
    MoveL Offs(pOrigin,377.08,80.44,0.00),v40,z0,tPen\WObj:=wPaper;
    MoveL Offs(pOrigin,382.81,79.38,0.00),v40,z0,tPen\WObj:=wPaper;
    MoveL Offs(pOrigin,387.91,77.89,0.00),v40,fine,tPen\WObj:=wPaper;
    MoveL Offs(pOrigin,387.91,77.89,6.00),v60,z5,tPen\WObj:=wPaper;
    MoveL Offs(pOrigin,384.94,85.11,6.00),vTravel,z5,tPen\WObj:=wPaper;
    MoveL Offs(pOrigin,384.94,85.11,0.00),v60,z0,tPen\WObj:=wPaper;
    MoveL Offs(pOrigin,381.96,85.11,0.00),v40,fine,tPen\WObj:=wPaper;
    MoveL Offs(pOrigin,381.96,85.11,6.00),v60,z5,tPen\WObj:=wPaper;
    MoveL Offs(pOrigin,378.35,87.03,6.00),vTravel,z5,tPen\WObj:=wPaper;
    MoveL Offs(pOrigin,378.35,87.03,0.00),v60,z0,tPen\WObj:=wPaper;
    MoveL Offs(pOrigin,381.75,88.51,0.00),v40,z0,tPen\WObj:=wPaper;
    MoveL Offs(pOrigin,387.06,89.79,0.00),v40,z0,tPen\WObj:=wPaper;
    MoveL Offs(pOrigin,391.10,90.00,0.00),v40,z0,tPen\WObj:=wPaper;
    MoveL Offs(pOrigin,397.05,89.15,0.00),v40,fine,tPen\WObj:=wPaper;
    MoveL Offs(pOrigin,397.05,89.15,6.00),v60,z5,tPen\WObj:=wPaper;
    MoveL Offs(pOrigin,404.06,80.65,6.00),vTravel,z5,tPen\WObj:=wPaper;
    MoveL Offs(pOrigin,404.06,80.65,0.00),v60,z0,tPen\WObj:=wPaper;
    MoveL Offs(pOrigin,404.49,80.44,0.00),v40,z0,tPen\WObj:=wPaper;
    MoveL Offs(pOrigin,404.06,80.65,0.00),v40,fine,tPen\WObj:=wPaper;
    MoveL Offs(pOrigin,404.06,80.65,6.00),v60,z5,tPen\WObj:=wPaper;
    MoveL Offs(pOrigin,405.76,79.16,6.00),vTravel,z5,tPen\WObj:=wPaper;
    MoveL Offs(pOrigin,405.76,79.16,0.00),v60,z0,tPen\WObj:=wPaper;
    MoveL Offs(pOrigin,405.55,79.59,0.00),v40,z0,tPen\WObj:=wPaper;
    MoveL Offs(pOrigin,405.76,79.16,0.00),v40,z0,tPen\WObj:=wPaper;
    MoveL Offs(pOrigin,405.12,78.31,0.00),v40,z0,tPen\WObj:=wPaper;
    MoveL Offs(pOrigin,404.70,78.74,0.00),v40,z0,tPen\WObj:=wPaper;
    MoveL Offs(pOrigin,405.12,78.31,0.00),v40,fine,tPen\WObj:=wPaper;
    MoveL Offs(pOrigin,405.12,78.31,6.00),v60,z5,tPen\WObj:=wPaper;
    MoveL Offs(pOrigin,406.40,77.68,6.00),vTravel,z5,tPen\WObj:=wPaper;
    MoveL Offs(pOrigin,406.40,77.68,0.00),v60,z0,tPen\WObj:=wPaper;
    MoveL Offs(pOrigin,406.61,77.25,0.00),v40,z0,tPen\WObj:=wPaper;
    MoveL Offs(pOrigin,407.60,76.90,0.00),v40,z0,tPen\WObj:=wPaper;
    MoveL Offs(pOrigin,407.60,77.68,0.00),v40,z0,tPen\WObj:=wPaper;
    MoveL Offs(pOrigin,406.61,78.03,0.00),v40,z0,tPen\WObj:=wPaper;
    MoveL Offs(pOrigin,406.40,77.68,0.00),v40,fine,tPen\WObj:=wPaper;
    MoveL Offs(pOrigin,406.40,77.68,6.00),v60,z5,tPen\WObj:=wPaper;
    MoveL Offs(pOrigin,407.67,76.82,6.00),vTravel,z5,tPen\WObj:=wPaper;
    MoveL Offs(pOrigin,407.67,76.82,0.00),v60,z0,tPen\WObj:=wPaper;
    MoveL Offs(pOrigin,411.50,72.57,0.00),v40,fine,tPen\WObj:=wPaper;
    MoveL Offs(pOrigin,411.50,72.57,6.00),v60,z5,tPen\WObj:=wPaper;
    MoveL Offs(pOrigin,410.01,74.28,6.00),vTravel,z5,tPen\WObj:=wPaper;
  ENDPROC

